LIN {X 0,Y 569.528,Z 1029.936,A -85,B 0,C 180,E1 26173.056,E2 26173.056} C_VEL
LIN {X 0,Y 570.393,Z 1020.294,A -85,B 0,C 180,E1 26170.971,E2 26170.971} C_VEL
LIN {X 0,Y 571.61,Z 1008.72,A -85,B 0,C 180,E1 26168.771,E2 26168.771} C_VEL
LIN {X 0,Y 573.314,Z 993.99,A -85,B 0,C 180,E1 26166.351,E2 26166.351} C_VEL
LIN {X 0,Y 575.02,Z 980.852,A -85,B 0,C 180,E1 26164.454,E2 26164.454} C_VEL
LIN {X 0,Y 577.029,Z 966.146,A -85,B 0,C 180,E1 26162.553,E2 26162.553} C_VEL
LIN {X 0,Y 579.743,Z 946.853,A -85,B 0,C 180,E1 26160.373,E2 26160.373} C_VEL
LIN {X 0,Y 582.096,Z 930.583,A -85,B 0,C 180,E1 26158.751,E2 26158.751} C_VEL
LIN {X 0,Y 584.678,Z 912.881,A -85,B 0,C 180,E1 26157.172,E2 26157.172} C_VEL
LIN {X 0,Y 587.865,Z 890.248,A -85,B 0,C 180,E1 26155.41,E2 26155.41} C_VEL
LIN {X 0,Y 590.454,Z 871.427,A -85,B 0,C 180,E1 26154.132,E2 26154.132} C_VEL
LIN {X 0,Y 593.347,Z 849.656,A -85,B 0,C 180,E1 26152.834,E2 26152.834} C_VEL
LIN {X 0,Y 596.171,Z 826.041,A -85,B 0,C 180,E1 26151.643,E2 26151.643} C_VEL
LIN {X 0,Y 598.242,Z 806.976,A -85,B 0,C 180,E1 26150.819,E2 26150.819} C_VEL
LIN {X 0,Y 600.276,Z 786.144,A -85,B 0,C 180,E1 26150.049,E2 26150.049} C_VEL
LIN {X 0,Y 602.478,Z 760.102,A -85,B 0,C 180,E1 26149.27,E2 26149.27} C_VEL
LIN {X 0,Y 603.931,Z 737.618,A -85,B 0,C 180,E1 26148.757,E2 26148.757} C_VEL
LIN {X 0,Y 604.964,Z 715.893,A -85,B 0,C 180,E1 26148.38,E2 26148.38} C_VEL
LIN {X 0,Y 610.807,Z 481.076,A -85,B 0,C 180,E1 26145.176,E2 26145.176} C_VEL
LIN {X 0,Y 614.185,Z 345.469,A -85,B 0,C 180,E1 26143.295,E2 26143.295} C_VEL
LIN {X 0,Y 598.706,Z 321.323,A -85,B 0,C 180,E1 26141.34,E2 26141.34} C_VEL
LIN {X 0,Y 585.115,Z 301.426,A -85,B 0,C 180,E1 26139.504,E2 26139.504} C_VEL
LIN {X 0,Y 575.623,Z 288.007,A -85,B 0,C 180,E1 26138.136,E2 26138.136} C_VEL
LIN {X 0,Y 573.982,Z 285.549,A -85,B 0,C 180,E1 26137.821,E2 26137.821} C_VEL
LIN {X 0,Y 570.798,Z 278.728,A -85,B 0,C 180,E1 26136.68,E2 26136.68} C_VEL
LIN {X 0,Y 569.328,Z 275.166,A -85,B 0,C 180,E1 26136.04,E2 26136.04} C_VEL
LIN {X 0,Y 569.375,Z 275.014,A -85,B 0,C 180,E1 26132.864,E2 26132.864} C_VEL
LIN {X 0,Y 569.308,Z 275.021,A -85,B 0,C 180,E1 26129.805,E2 26129.805} C_VEL
LIN {X 0,Y 569.365,Z 275.04,A -85,B 0,C 180,E1 26126.604,E2 26126.604} C_VEL
LIN {X 0,Y 569.315,Z 275.047,A -85,B 0,C 180,E1 26123.496,E2 26123.496} C_VEL
LIN {X 0,Y 569.337,Z 275.044,A -85,B 0,C 180,E1 26120.242,E2 26120.242} C_VEL
LIN {X 0,Y 569.33,Z 275.049,A -85,B 0,C 180,E1 26117.161,E2 26117.161} C_VEL
LIN {X 0,Y 569.315,Z 275.058,A -85,B 0,C 180,E1 26113.819,E2 26113.819} C_VEL
LIN {X 0,Y 569.363,Z 275.057,A -85,B 0,C 180,E1 26110.728,E2 26110.728} C_VEL
LIN {X 0,Y 569.31,Z 275.052,A -85,B 0,C 180,E1 26107.569,E2 26107.569} C_VEL
LIN {X 0,Y 569.374,Z 275.038,A -85,B 0,C 180,E1 26104.432,E2 26104.432} C_VEL
LIN {X 0,Y 569.31,Z 275.06,A -85,B 0,C 180,E1 26101.308,E2 26101.308} C_VEL
LIN {X 0,Y 569.37,Z 275.055,A -85,B 0,C 180,E1 26098.189,E2 26098.189} C_VEL
LIN {X 0,Y 569.312,Z 275.045,A -85,B 0,C 180,E1 26095.063,E2 26095.063} C_VEL
LIN {X 0,Y 569.341,Z 275.041,A -85,B 0,C 180,E1 26091.822,E2 26091.822} C_VEL
LIN {X 0,Y 569.326,Z 275.062,A -85,B 0,C 180,E1 26088.758,E2 26088.758} C_VEL
LIN {X 0,Y 569.318,Z 275.065,A -85,B 0,C 180,E1 26085.401,E2 26085.401} C_VEL
LIN {X 0,Y 569.356,Z 275.041,A -85,B 0,C 180,E1 26082.313,E2 26082.313} C_VEL
LIN {X 0,Y 569.31,Z 275.043,A -85,B 0,C 180,E1 26079.112,E2 26079.112} C_VEL
LIN {X 0,Y 569.372,Z 275.038,A -85,B 0,C 180,E1 26076.067,E2 26076.067} C_VEL
LIN {X 0,Y 569.302,Z 274.992,A -85,B 0,C 180,E1 26072.829,E2 26072.829} C_VEL
LIN {X 0,Y 569.376,Z 275.054,A -85,B 0,C 180,E1 26069.734,E2 26069.734} C_VEL
LIN {X 0,Y 569.309,Z 274.991,A -85,B 0,C 180,E1 26066.531,E2 26066.531} C_VEL
LIN {X 0,Y 569.327,Z 275.051,A -85,B 0,C 180,E1 26063.21,E2 26063.21} C_VEL
LIN {X 0,Y 569.336,Z 275.11,A -85,B 0,C 180,E1 26060.201,E2 26060.201} C_VEL
LIN {X 0,Y 570.614,Z 278.424,A -85,B 0,C 180,E1 26059.582,E2 26059.582} C_VEL
LIN {X 0,Y 571.787,Z 280.362,A -85,B 0,C 180,E1 26059.303,E2 26059.303} C_VEL
LIN {X 0,Y 575.084,Z 284.719,A -85,B 0,C 180,E1 26058.812,E2 26058.812} C_VEL
LIN {X 0,Y 589.505,Z 304.979,A -85,B 0,C 180,E1 26056.761,E2 26056.761} C_VEL
LIN {X 0,Y 601.117,Z 322.104,A -85,B 0,C 180,E1 26055.215,E2 26055.215} C_VEL
LIN {X 0,Y 614.233,Z 342.476,A -85,B 0,C 180,E1 26053.57,E2 26053.57} C_VEL
LIN {X 0,Y 609.182,Z 540.418,A -85,B 0,C 180,E1 26050.843,E2 26050.843} C_VEL
LIN {X 0,Y 608.261,Z 548.118,A -85,B 0,C 180,E1 26050.802,E2 26050.802} C_VEL
LIN {X 0,Y 603.163,Z 568.707,A -85,B 0,C 180,E1 26050.927,E2 26050.927} C_VEL
LIN {X 0,Y 602.444,Z 575.314,A -85,B 0,C 180,E1 26050.885,E2 26050.885} C_VEL
LIN {X 0,Y 598.824,Z 711.721,A -85,B 0,C 180,E1 26049.003,E2 26049.003} C_VEL
LIN {X 0,Y 597.3,Z 738.812,A -85,B 0,C 180,E1 26048.485,E2 26048.485} C_VEL
LIN {X 0,Y 595.509,Z 762.096,A -85,B 0,C 180,E1 26047.873,E2 26047.873} C_VEL
LIN {X 0,Y 593.502,Z 784.135,A -85,B 0,C 180,E1 26047.155,E2 26047.155} C_VEL
LIN {X 0,Y 590.692,Z 810.488,A -85,B 0,C 180,E1 26046.091,E2 26046.091} C_VEL
LIN {X 0,Y 588.249,Z 830.386,A -85,B 0,C 180,E1 26045.131,E2 26045.131} C_VEL
LIN {X 0,Y 585.686,Z 849.812,A -85,B 0,C 180,E1 26044.053,E2 26044.053} C_VEL
LIN {X 0,Y 582.368,Z 873.343,A -85,B 0,C 180,E1 26042.539,E2 26042.539} C_VEL
LIN {X 0,Y 579.492,Z 892.375,A -85,B 0,C 180,E1 26041.122,E2 26041.122} C_VEL
LIN {X 0,Y 576.819,Z 909.782,A -85,B 0,C 180,E1 26039.663,E2 26039.663} C_VEL
LIN {X 0,Y 573.672,Z 930.084,A -85,B 0,C 180,E1 26037.734,E2 26037.734} C_VEL
LIN {X 0,Y 571.147,Z 946.426,A -85,B 0,C 180,E1 26035.955,E2 26035.955} C_VEL
LIN {X 0,Y 568.951,Z 961.1,A -85,B 0,C 180,E1 26034.172,E2 26034.172} C_VEL
LIN {X 0,Y 566.637,Z 977.255,A -85,B 0,C 180,E1 26031.968,E2 26031.968} C_VEL
LIN {X 0,Y 564.777,Z 991.296,A -85,B 0,C 180,E1 26029.764,E2 26029.764} C_VEL
LIN {X 0,Y 563.414,Z 1002.582,A -85,B 0,C 180,E1 26027.773,E2 26027.773} C_VEL
LIN {X 0,Y 562.168,Z 1014.61,A -85,B 0,C 180,E1 26025.368,E2 26025.368} C_VEL
LIN {X 0,Y 561.216,Z 1025.111,A -85,B 0,C 180,E1 26022.868,E2 26022.868} C_VEL
LIN {X 0,Y 560.704,Z 1032.614,A -85,B 0,C 180,E1 26020.792,E2 26020.792} C_VEL
LIN {X 0,Y 560.275,Z 1040.198,A -85,B 0,C 180,E1 26018.311,E2 26018.311} C_VEL
LIN {X 0,Y 560.033,Z 1046.307,A -85,B 0,C 180,E1 26015.738,E2 26015.738} C_VEL
LIN {X 0,Y 559.954,Z 1050.223,A -85,B 0,C 180,E1 26013.583,E2 26013.583} C_VEL
LIN {X 0,Y 559.903,Z 1053.047,A -85,B 0,C 180,E1 26011.433,E2 26011.433} C_VEL
LIN {X 0,Y 559.908,Z 1054.995,A -85,B 0,C 180,E1 26008.977,E2 26008.977} C_VEL
LIN {X 0,Y 559.892,Z 1055.388,A -85,B 0,C 180,E1 26006.416,E2 26006.416} C_VEL
LIN {X 0,Y 559.915,Z 1054.551,A -85,B 0,C 180,E1 26004.261,E2 26004.261} C_VEL
LIN {X 0,Y 559.907,Z 1052.74,A -85,B 0,C 180,E1 26002.2,E2 26002.2} C_VEL
LIN {X 0,Y 559.967,Z 1049.596,A -85,B 0,C 180,E1 25999.922,E2 25999.922} C_VEL
LIN {X 0,Y 560.103,Z 1044.215,A -85,B 0,C 180,E1 25997.211,E2 25997.211} C_VEL
LIN {X 0,Y 560.378,Z 1038.165,A -85,B 0,C 180,E1 25994.9,E2 25994.9} C_VEL
LIN {X 0,Y 560.79,Z 1031.129,A -85,B 0,C 180,E1 25992.677,E2 25992.677} C_VEL
LIN {X 0,Y 561.572,Z 1020.991,A -85,B 0,C 180,E1 25990.01,E2 25990.01} C_VEL
LIN {X 0,Y 562.532,Z 1010.781,A -85,B 0,C 180,E1 25987.753,E2 25987.753} C_VEL
LIN {X 0,Y 563.698,Z 1000.216,A -85,B 0,C 180,E1 25985.7,E2 25985.7} C_VEL
LIN {X 0,Y 565.513,Z 985.511,A -85,B 0,C 180,E1 25983.201,E2 25983.201} C_VEL
LIN {X 0,Y 567.441,Z 971.489,A -85,B 0,C 180,E1 25981.131,E2 25981.131} C_VEL
LIN {X 0,Y 569.484,Z 957.456,A -85,B 0,C 180,E1 25979.274,E2 25979.274} C_VEL
LIN {X 0,Y 572.415,Z 938.223,A -85,B 0,C 180,E1 25977.035,E2 25977.035} C_VEL
LIN {X 0,Y 574.992,Z 921.578,A -85,B 0,C 180,E1 25975.339,E2 25975.339} C_VEL
LIN {X 0,Y 577.583,Z 904.918,A -85,B 0,C 180,E1 25973.82,E2 25973.82} C_VEL
LIN {X 0,Y 580.874,Z 883.291,A -85,B 0,C 180,E1 25972.083,E2 25972.083} C_VEL
LIN {X 0,Y 583.821,Z 863.031,A -85,B 0,C 180,E1 25970.678,E2 25970.678} C_VEL
LIN {X 0,Y 586.657,Z 842.71,A -85,B 0,C 180,E1 25969.442,E2 25969.442} C_VEL
LIN {X 0,Y 589.839,Z 817.959,A -85,B 0,C 180,E1 25968.16,E2 25968.16} C_VEL
LIN {X 0,Y 592.189,Z 797.521,A -85,B 0,C 180,E1 25967.264,E2 25967.264} C_VEL
LIN {X 0,Y 594.25,Z 777.464,A -85,B 0,C 180,E1 25966.514,E2 25966.514} C_VEL
LIN {X 0,Y 596.578,Z 751.419,A -85,B 0,C 180,E1 25965.722,E2 25965.722} C_VEL
LIN {X 0,Y 598.111,Z 728.952,A -85,B 0,C 180,E1 25965.2,E2 25965.2} C_VEL
LIN {X 0,Y 599.204,Z 707.344,A -85,B 0,C 180,E1 25964.818,E2 25964.818} C_VEL
LIN {X 0,Y 605.825,Z 470.078,A -85,B 0,C 180,E1 25961.519,E2 25961.519} C_VEL
LIN {X 0,Y 609.288,Z 345.786,A -85,B 0,C 180,E1 25959.748,E2 25959.748} C_VEL
LIN {X 0,Y 596.939,Z 326.269,A -85,B 0,C 180,E1 25958.04,E2 25958.04} C_VEL
LIN {X 0,Y 582.975,Z 306.239,A -85,B 0,C 180,E1 25955.976,E2 25955.976} C_VEL
LIN {X 0,Y 575.262,Z 295.929,A -85,B 0,C 180,E1 25954.758,E2 25954.758} C_VEL
LIN {X 0,Y 570.969,Z 290.29,A -85,B 0,C 180,E1 25954.053,E2 25954.053} C_VEL
LIN {X 0,Y 567.524,Z 285.647,A -85,B 0,C 180,E1 25953.467,E2 25953.467} C_VEL
LIN {X 0,Y 564.242,Z 281.388,A -85,B 0,C 180,E1 25952.898,E2 25952.898} C_VEL
LIN {X 0,Y 562.325,Z 278.884,A -85,B 0,C 180,E1 25952.48,E2 25952.48} C_VEL
LIN {X 0,Y 561.444,Z 276.206,A -85,B 0,C 180,E1 25951.934,E2 25951.934} C_VEL
LIN {X 0,Y 561.373,Z 276.043,A -85,B 0,C 180,E1 25948.978,E2 25948.978} C_VEL
LIN {X 0,Y 561.403,Z 275.99,A -85,B 0,C 180,E1 25945.759,E2 25945.759} C_VEL
LIN {X 0,Y 561.383,Z 276.054,A -85,B 0,C 180,E1 25942.689,E2 25942.689} C_VEL
LIN {X 0,Y 561.372,Z 275.997,A -85,B 0,C 180,E1 25939.239,E2 25939.239} C_VEL
LIN {X 0,Y 561.423,Z 276.037,A -85,B 0,C 180,E1 25936.131,E2 25936.131} C_VEL
LIN {X 0,Y 561.365,Z 275.993,A -85,B 0,C 180,E1 25932.969,E2 25932.969} C_VEL
LIN {X 0,Y 561.435,Z 276.039,A -85,B 0,C 180,E1 25929.741,E2 25929.741} C_VEL
LIN {X 0,Y 561.364,Z 275.982,A -85,B 0,C 180,E1 25926.648,E2 25926.648} C_VEL
LIN {X 0,Y 561.409,Z 276.047,A -85,B 0,C 180,E1 25923.369,E2 25923.369} C_VEL
LIN {X 0,Y 561.374,Z 275.984,A -85,B 0,C 180,E1 25920.306,E2 25920.306} C_VEL
LIN {X 0,Y 561.383,Z 276.051,A -85,B 0,C 180,E1 25916.937,E2 25916.937} C_VEL
LIN {X 0,Y 561.416,Z 275.981,A -85,B 0,C 180,E1 25913.763,E2 25913.763} C_VEL
LIN {X 0,Y 561.37,Z 276.036,A -85,B 0,C 180,E1 25910.569,E2 25910.569} C_VEL
LIN {X 0,Y 561.429,Z 275.989,A -85,B 0,C 180,E1 25907.346,E2 25907.346} C_VEL
LIN {X 0,Y 561.369,Z 276.019,A -85,B 0,C 180,E1 25904.292,E2 25904.292} C_VEL
LIN {X 0,Y 561.41,Z 276.002,A -85,B 0,C 180,E1 25901.036,E2 25901.036} C_VEL
LIN {X 0,Y 561.381,Z 276.02,A -85,B 0,C 180,E1 25897.925,E2 25897.925} C_VEL
LIN {X 0,Y 561.381,Z 276.036,A -85,B 0,C 180,E1 25894.559,E2 25894.559} C_VEL
LIN {X 0,Y 561.414,Z 276.032,A -85,B 0,C 180,E1 25891.49,E2 25891.49} C_VEL
LIN {X 0,Y 561.368,Z 275.993,A -85,B 0,C 180,E1 25888.302,E2 25888.302} C_VEL
LIN {X 0,Y 561.409,Z 276.234,A -85,B 0,C 180,E1 25885.778,E2 25885.778} C_VEL
LIN {X 0,Y 563.065,Z 279.972,A -85,B 0,C 180,E1 25884.999,E2 25884.999} C_VEL
LIN {X 0,Y 566.244,Z 286.174,A -85,B 0,C 180,E1 25883.813,E2 25883.813} C_VEL
LIN {X 0,Y 577.941,Z 302.001,A -85,B 0,C 180,E1 25881.856,E2 25881.856} C_VEL
LIN {X 0,Y 588.085,Z 316.172,A -85,B 0,C 180,E1 25880.292,E2 25880.292} C_VEL
LIN {X 0,Y 599.299,Z 332.935,A -85,B 0,C 180,E1 25878.662,E2 25878.662} C_VEL
LIN {X 0,Y 609.505,Z 349.548,A -85,B 0,C 180,E1 25877.259,E2 25877.259} C_VEL
LIN {X 0,Y 602.826,Z 581.277,A -85,B 0,C 180,E1 25874.013,E2 25874.013} C_VEL
LIN {X 0,Y 598.937,Z 720.481,A -85,B 0,C 180,E1 25872.074,E2 25872.074} C_VEL
LIN {X 0,Y 597.342,Z 747.614,A -85,B 0,C 180,E1 25871.554,E2 25871.554} C_VEL
LIN {X 0,Y 595.485,Z 771.005,A -85,B 0,C 180,E1 25870.937,E2 25870.937} C_VEL
LIN {X 0,Y 593.458,Z 792.738,A -85,B 0,C 180,E1 25870.227,E2 25870.227} C_VEL
LIN {X 0,Y 590.584,Z 819.273,A -85,B 0,C 180,E1 25869.157,E2 25869.157} C_VEL
LIN {X 0,Y 588.069,Z 839.646,A -85,B 0,C 180,E1 25868.174,E2 25868.174} C_VEL
LIN {X 0,Y 585.356,Z 860.369,A -85,B 0,C 180,E1 25867.022,E2 25867.022} C_VEL
LIN {X 0,Y 581.977,Z 884.248,A -85,B 0,C 180,E1 25865.474,E2 25865.474} C_VEL
LIN {X 0,Y 579.28,Z 902.355,A -85,B 0,C 180,E1 25864.123,E2 25864.123} C_VEL
LIN {X 0,Y 576.588,Z 920.113,A -85,B 0,C 180,E1 25862.637,E2 25862.637} C_VEL
LIN {X 0,Y 573.347,Z 941.298,A -85,B 0,C 180,E1 25860.613,E2 25860.613} C_VEL
LIN {X 0,Y 570.932,Z 957.248,A -85,B 0,C 180,E1 25858.876,E2 25858.876} C_VEL
LIN {X 0,Y 568.653,Z 972.852,A -85,B 0,C 180,E1 25856.978,E2 25856.978} C_VEL
LIN {X 0,Y 566.284,Z 989.784,A -85,B 0,C 180,E1 25854.627,E2 25854.627} C_VEL
LIN {X 0,Y 564.612,Z 1002.542,A -85,B 0,C 180,E1 25852.6,E2 25852.6} C_VEL
LIN {X 0,Y 563.112,Z 1015.592,A -85,B 0,C 180,E1 25850.258,E2 25850.258} C_VEL
LIN {X 0,Y 561.91,Z 1027.179,A -85,B 0,C 180,E1 25847.822,E2 25847.822} C_VEL
LIN {X 0,Y 561.157,Z 1035.877,A -85,B 0,C 180,E1 25845.714,E2 25845.714} C_VEL
LIN {X 0,Y 560.633,Z 1043.715,A -85,B 0,C 180,E1 25843.511,E2 25843.511} C_VEL
LIN {X 0,Y 560.216,Z 1051.623,A -85,B 0,C 180,E1 25840.801,E2 25840.801} C_VEL
LIN {X 0,Y 560.022,Z 1056.828,A -85,B 0,C 180,E1 25838.522,E2 25838.522} C_VEL
LIN {X 0,Y 559.955,Z 1060.486,A -85,B 0,C 180,E1 25836.459,E2 25836.459} C_VEL
LIN {X 0,Y 559.914,Z 1063.47,A -85,B 0,C 180,E1 25834.096,E2 25834.096} C_VEL
LIN {X 0,Y 559.9,Z 1065.19,A -85,B 0,C 180,E1 25831.433,E2 25831.433} C_VEL
LIN {X 0,Y 559.898,Z 1065.349,A -85,B 0,C 180,E1 25829.284,E2 25829.284} C_VEL
LIN {X 0,Y 559.913,Z 1064.436,A -85,B 0,C 180,E1 25827.134,E2 25827.134} C_VEL
LIN {X 0,Y 559.918,Z 1062.446,A -85,B 0,C 180,E1 25824.98,E2 25824.98} C_VEL
LIN {X 0,Y 559.999,Z 1058.461,A -85,B 0,C 180,E1 25822.294,E2 25822.294} C_VEL
LIN {X 0,Y 560.127,Z 1053.403,A -85,B 0,C 180,E1 25819.925,E2 25819.925} C_VEL
LIN {X 0,Y 560.387,Z 1047.876,A -85,B 0,C 180,E1 25817.846,E2 25817.846} C_VEL
LIN {X 0,Y 560.832,Z 1040.535,A -85,B 0,C 180,E1 25815.546,E2 25815.546} C_VEL
LIN {X 0,Y 561.656,Z 1029.935,A -85,B 0,C 180,E1 25812.811,E2 25812.811} C_VEL
LIN {X 0,Y 562.582,Z 1020.281,A -85,B 0,C 180,E1 25810.694,E2 25810.694} C_VEL
LIN {X 0,Y 563.89,Z 1008.718,A -85,B 0,C 180,E1 25808.466,E2 25808.466} C_VEL
LIN {X 0,Y 565.711,Z 993.988,A -85,B 0,C 180,E1 25806.014,E2 25806.014} C_VEL
LIN {X 0,Y 567.513,Z 980.818,A -85,B 0,C 180,E1 25804.091,E2 25804.091} C_VEL
LIN {X 0,Y 569.76,Z 965.215,A -85,B 0,C 180,E1 25802.059,E2 25802.059} C_VEL
LIN {X 0,Y 572.576,Z 946.397,A -85,B 0,C 180,E1 25799.922,E2 25799.922} C_VEL
LIN {X 0,Y 575.002,Z 930.5,A -85,B 0,C 180,E1 25798.321,E2 25798.321} C_VEL
LIN {X 0,Y 577.81,Z 912.188,A -85,B 0,C 180,E1 25796.673,E2 25796.673} C_VEL
LIN {X 0,Y 581.131,Z 889.829,A -85,B 0,C 180,E1 25794.923,E2 25794.923} C_VEL
LIN {X 0,Y 583.806,Z 871.342,A -85,B 0,C 180,E1 25793.659,E2 25793.659} C_VEL
LIN {X 0,Y 586.842,Z 849.57,A -85,B 0,C 180,E1 25792.351,E2 25792.351} C_VEL
LIN {X 0,Y 589.796,Z 825.94,A -85,B 0,C 180,E1 25791.152,E2 25791.152} C_VEL
LIN {X 0,Y 591.962,Z 806.826,A -85,B 0,C 180,E1 25790.321,E2 25790.321} C_VEL
LIN {X 0,Y 594.004,Z 786.663,A -85,B 0,C 180,E1 25789.572,E2 25789.572} C_VEL
LIN {X 0,Y 596.265,Z 761.264,A -85,B 0,C 180,E1 25788.801,E2 25788.801} C_VEL
LIN {X 0,Y 597.85,Z 737.716,A -85,B 0,C 180,E1 25788.258,E2 25788.258} C_VEL
LIN {X 0,Y 598.921,Z 716.111,A -85,B 0,C 180,E1 25787.88,E2 25787.88} C_VEL
LIN {X 0,Y 604.999,Z 482.812,A -85,B 0,C 180,E1 25784.673,E2 25784.673} C_VEL
LIN {X 0,Y 608.49,Z 349.049,A -85,B 0,C 180,E1 25782.803,E2 25782.803} C_VEL
LIN {X 0,Y 593.069,Z 324.968,A -85,B 0,C 180,E1 25780.808,E2 25780.808} C_VEL
LIN {X 0,Y 578.742,Z 303.894,A -85,B 0,C 180,E1 25778.812,E2 25778.812} C_VEL
LIN {X 0,Y 567.989,Z 289.037,A -85,B 0,C 180,E1 25777.207,E2 25777.207} C_VEL
LIN {X 0,Y 565.798,Z 285.613,A -85,B 0,C 180,E1 25776.805,E2 25776.805} C_VEL
LIN {X 0,Y 562.526,Z 279.268,A -85,B 0,C 180,E1 25775.663,E2 25775.663} C_VEL
LIN {X 0,Y 561.444,Z 276.151,A -85,B 0,C 180,E1 25775.098,E2 25775.098} C_VEL
LIN {X 0,Y 561.372,Z 276.039,A -85,B 0,C 180,E1 25771.938,E2 25771.938} C_VEL
LIN {X 0,Y 561.437,Z 275.984,A -85,B 0,C 180,E1 25768.741,E2 25768.741} C_VEL
LIN {X 0,Y 561.379,Z 276.053,A -85,B 0,C 180,E1 25765.533,E2 25765.533} C_VEL
LIN {X 0,Y 561.39,Z 276.053,A -85,B 0,C 180,E1 25762.156,E2 25762.156} C_VEL
LIN {X 0,Y 561.396,Z 276.044,A -85,B 0,C 180,E1 25759.13,E2 25759.13} C_VEL
LIN {X 0,Y 561.374,Z 276.039,A -85,B 0,C 180,E1 25755.814,E2 25755.814} C_VEL
LIN {X 0,Y 561.424,Z 276.028,A -85,B 0,C 180,E1 25752.759,E2 25752.759} C_VEL
LIN {X 0,Y 561.371,Z 276.046,A -85,B 0,C 180,E1 25749.535,E2 25749.535} C_VEL
LIN {X 0,Y 561.438,Z 276.048,A -85,B 0,C 180,E1 25746.339,E2 25746.339} C_VEL
LIN {X 0,Y 561.376,Z 276.042,A -85,B 0,C 180,E1 25743.165,E2 25743.165} C_VEL
LIN {X 0,Y 561.387,Z 276.03,A -85,B 0,C 180,E1 25739.796,E2 25739.796} C_VEL
LIN {X 0,Y 561.399,Z 276.043,A -85,B 0,C 180,E1 25736.733,E2 25736.733} C_VEL
LIN {X 0,Y 561.375,Z 276.052,A -85,B 0,C 180,E1 25733.454,E2 25733.454} C_VEL
LIN {X 0,Y 561.426,Z 276.03,A -85,B 0,C 180,E1 25730.363,E2 25730.363} C_VEL
LIN {X 0,Y 561.368,Z 276.03,A -85,B 0,C 180,E1 25727.135,E2 25727.135} C_VEL
LIN {X 0,Y 561.434,Z 276.032,A -85,B 0,C 180,E1 25723.975,E2 25723.975} C_VEL
LIN {X 0,Y 561.379,Z 276.052,A -85,B 0,C 180,E1 25720.761,E2 25720.761} C_VEL
LIN {X 0,Y 561.382,Z 276.053,A -85,B 0,C 180,E1 25717.311,E2 25717.311} C_VEL
LIN {X 0,Y 561.401,Z 275.973,A -85,B 0,C 180,E1 25714.241,E2 25714.241} C_VEL
LIN {X 0,Y 561.37,Z 276.035,A -85,B 0,C 180,E1 25710.991,E2 25710.991} C_VEL
LIN {X 0,Y 561.425,Z 275.982,A -85,B 0,C 180,E1 25707.945,E2 25707.945} C_VEL
LIN {X 0,Y 561.369,Z 276.023,A -85,B 0,C 180,E1 25704.753,E2 25704.753} C_VEL
LIN {X 0,Y 561.429,Z 276.025,A -85,B 0,C 180,E1 25701.57,E2 25701.57} C_VEL
LIN {X 0,Y 561.421,Z 276.33,A -85,B 0,C 180,E1 25701.064,E2 25701.064} C_VEL
LIN {X 0,Y 562.725,Z 279.607,A -85,B 0,C 180,E1 25700.497,E2 25700.497} C_VEL
LIN {X 0,Y 568.48,Z 287.302,A -85,B 0,C 180,E1 25699.581,E2 25699.581} C_VEL
LIN {X 0,Y 579.175,Z 301.934,A -85,B 0,C 180,E1 25697.995,E2 25697.995} C_VEL
LIN {X 0,Y 592.975,Z 321.874,A -85,B 0,C 180,E1 25696.078,E2 25696.078} C_VEL
LIN {X 0,Y 608.546,Z 345.901,A -85,B 0,C 180,E1 25694.064,E2 25694.064} C_VEL
LIN {X 0,Y 602.665,Z 566.89,A -85,B 0,C 180,E1 25691,E2 25691} C_VEL
LIN {X 0,Y 602.444,Z 575.314,A -85,B 0,C 180,E1 25690.885,E2 25690.885} C_VEL
LIN {X 0,Y 601.525,Z 583.011,A -85,B 0,C 180,E1 25690.844,E2 25690.844} C_VEL
LIN {X 0,Y 596.424,Z 603.594,A -85,B 0,C 180,E1 25690.97,E2 25690.97} C_VEL
LIN {X 0,Y 595.678,Z 610.202,A -85,B 0,C 180,E1 25690.931,E2 25690.931} C_VEL
LIN {X 0,Y 592.806,Z 712.303,A -85,B 0,C 180,E1 25689.507,E2 25689.507} C_VEL
LIN {X 0,Y 591.143,Z 740.202,A -85,B 0,C 180,E1 25688.962,E2 25688.962} C_VEL
LIN {X 0,Y 589.328,Z 762.839,A -85,B 0,C 180,E1 25688.36,E2 25688.36} C_VEL
LIN {X 0,Y 587.139,Z 785.951,A -85,B 0,C 180,E1 25687.596,E2 25687.596} C_VEL
LIN {X 0,Y 584.41,Z 810.278,A -85,B 0,C 180,E1 25686.602,E2 25686.602} C_VEL
LIN {X 0,Y 581.833,Z 830.487,A -85,B 0,C 180,E1 25685.623,E2 25685.623} C_VEL
LIN {X 0,Y 579.156,Z 849.987,A -85,B 0,C 180,E1 25684.535,E2 25684.535} C_VEL
LIN {X 0,Y 575.693,Z 873.47,A -85,B 0,C 180,E1 25683.012,E2 25683.012} C_VEL
LIN {X 0,Y 572.691,Z 892.433,A -85,B 0,C 180,E1 25681.586,E2 25681.586} C_VEL
LIN {X 0,Y 569.895,Z 909.784,A -85,B 0,C 180,E1 25680.118,E2 25680.118} C_VEL
LIN {X 0,Y 566.565,Z 930.101,A -85,B 0,C 180,E1 25678.17,E2 25678.17} C_VEL
LIN {X 0,Y 563.824,Z 946.901,A -85,B 0,C 180,E1 25676.318,E2 25676.318} C_VEL
LIN {X 0,Y 561.5,Z 961.649,A -85,B 0,C 180,E1 25674.499,E2 25674.499} C_VEL
LIN {X 0,Y 558.959,Z 978.32,A -85,B 0,C 180,E1 25672.175,E2 25672.175} C_VEL
LIN {X 0,Y 557.094,Z 991.586,A -85,B 0,C 180,E1 25670.048,E2 25670.048} C_VEL
LIN {X 0,Y 555.579,Z 1003.394,A -85,B 0,C 180,E1 25667.924,E2 25667.924} C_VEL
LIN {X 0,Y 554.167,Z 1016.175,A -85,B 0,C 180,E1 25665.274,E2 25665.274} C_VEL
LIN {X 0,Y 553.309,Z 1025.285,A -85,B 0,C 180,E1 25663.055,E2 25663.055} C_VEL
LIN {X 0,Y 552.734,Z 1033.114,A -85,B 0,C 180,E1 25660.844,E2 25660.844} C_VEL
LIN {X 0,Y 552.272,Z 1040.877,A -85,B 0,C 180,E1 25658.223,E2 25658.223} C_VEL
LIN {X 0,Y 552.036,Z 1046.6,A -85,B 0,C 180,E1 25655.717,E2 25655.717} C_VEL
LIN {X 0,Y 551.957,Z 1050.291,A -85,B 0,C 180,E1 25653.635,E2 25653.635} C_VEL
LIN {X 0,Y 551.903,Z 1053.095,A -85,B 0,C 180,E1 25651.453,E2 25651.453} C_VEL
LIN {X 0,Y 551.908,Z 1055.024,A -85,B 0,C 180,E1 25648.962,E2 25648.962} C_VEL
LIN {X 0,Y 551.893,Z 1055.378,A -85,B 0,C 180,E1 25646.364,E2 25646.364} C_VEL
LIN {X 0,Y 551.915,Z 1054.521,A -85,B 0,C 180,E1 25644.177,E2 25644.177} C_VEL
LIN {X 0,Y 551.912,Z 1052.691,A -85,B 0,C 180,E1 25642.086,E2 25642.086} C_VEL
LIN {X 0,Y 551.977,Z 1049.527,A -85,B 0,C 180,E1 25639.774,E2 25639.774} C_VEL
LIN {X 0,Y 552.123,Z 1044.017,A -85,B 0,C 180,E1 25636.987,E2 25636.987} C_VEL
LIN {X 0,Y 552.409,Z 1038.227,A -85,B 0,C 180,E1 25634.745,E2 25634.745} C_VEL
LIN {X 0,Y 552.844,Z 1031.33,A -85,B 0,C 180,E1 25632.529,E2 25632.529} C_VEL
LIN {X 0,Y 553.649,Z 1021.605,A -85,B 0,C 180,E1 25629.905,E2 25629.905} C_VEL
LIN {X 0,Y 554.698,Z 1011.073,A -85,B 0,C 180,E1 25627.533,E2 25627.533} C_VEL
LIN {X 0,Y 555.938,Z 1000.54,A -85,B 0,C 180,E1 25625.451,E2 25625.451} C_VEL
LIN {X 0,Y 557.87,Z 985.954,A -85,B 0,C 180,E1 25622.919,E2 25622.919} C_VEL
LIN {X 0,Y 559.902,Z 972.006,A -85,B 0,C 180,E1 25620.822,E2 25620.822} C_VEL
LIN {X 0,Y 562.054,Z 958.016,A -85,B 0,C 180,E1 25618.942,E2 25618.942} C_VEL
LIN {X 0,Y 564.988,Z 939.912,A -85,B 0,C 180,E1 25616.788,E2 25616.788} C_VEL
LIN {X 0,Y 567.85,Z 922.304,A -85,B 0,C 180,E1 25614.964,E2 25614.964} C_VEL
LIN {X 0,Y 570.56,Z 905.692,A -85,B 0,C 180,E1 25613.428,E2 25613.428} C_VEL
LIN {X 0,Y 574.012,Z 884.213,A -85,B 0,C 180,E1 25611.675,E2 25611.675} C_VEL
LIN {X 0,Y 577.093,Z 864.052,A -85,B 0,C 180,E1 25610.258,E2 25610.258} C_VEL
LIN {X 0,Y 579.998,Z 844.262,A -85,B 0,C 180,E1 25609.034,E2 25609.034} C_VEL
LIN {X 0,Y 583.387,Z 819.502,A -85,B 0,C 180,E1 25607.723,E2 25607.723} C_VEL
LIN {X 0,Y 585.857,Z 799.097,A -85,B 0,C 180,E1 25606.812,E2 25606.812} C_VEL
LIN {X 0,Y 588.053,Z 778.788,A -85,B 0,C 180,E1 25606.04,E2 25606.04} C_VEL
LIN {X 0,Y 590.445,Z 753.849,A -85,B 0,C 180,E1 25605.26,E2 25605.26} C_VEL
LIN {X 0,Y 592.19,Z 729.486,A -85,B 0,C 180,E1 25604.684,E2 25604.684} C_VEL
LIN {X 0,Y 593.34,Z 707.825,A -85,B 0,C 180,E1 25604.297,E2 25604.297} C_VEL
LIN {X 0,Y 600.267,Z 471.875,A -85,B 0,C 180,E1 25600.989,E2 25600.989} C_VEL
LIN {X 0,Y 603.887,Z 349.551,A -85,B 0,C 180,E1 25599.235,E2 25599.235} C_VEL
LIN {X 0,Y 591.822,Z 330.448,A -85,B 0,C 180,E1 25597.522,E2 25597.522} C_VEL
LIN {X 0,Y 578.691,Z 311.617,A -85,B 0,C 180,E1 25595.532,E2 25595.532} C_VEL
LIN {X 0,Y 571.67,Z 302.16,A -85,B 0,C 180,E1 25594.399,E2 25594.399} C_VEL
LIN {X 0,Y 564.132,Z 292.127,A -85,B 0,C 180,E1 25593.117,E2 25593.117} C_VEL
LIN {X 0,Y 556.065,Z 282.011,A -85,B 0,C 180,E1 25591.673,E2 25591.673} C_VEL
LIN {X 0,Y 553.925,Z 278.958,A -85,B 0,C 180,E1 25591.173,E2 25591.173} C_VEL
LIN {X 0,Y 553.457,Z 277.112,A -85,B 0,C 180,E1 25590.749,E2 25590.749} C_VEL
LIN {X 0,Y 553.439,Z 277.008,A -85,B 0,C 180,E1 25587.433,E2 25587.433} C_VEL
LIN {X 0,Y 553.485,Z 276.999,A -85,B 0,C 180,E1 25584.21,E2 25584.21} C_VEL
LIN {X 0,Y 553.429,Z 276.99,A -85,B 0,C 180,E1 25581.072,E2 25581.072} C_VEL
LIN {X 0,Y 553.492,Z 277.017,A -85,B 0,C 180,E1 25577.819,E2 25577.819} C_VEL
LIN {X 0,Y 553.431,Z 276.983,A -85,B 0,C 180,E1 25574.652,E2 25574.652} C_VEL
LIN {X 0,Y 553.447,Z 277.026,A -85,B 0,C 180,E1 25571.252,E2 25571.252} C_VEL
LIN {X 0,Y 553.466,Z 276.976,A -85,B 0,C 180,E1 25568.106,E2 25568.106} C_VEL
LIN {X 0,Y 553.432,Z 277.011,A -85,B 0,C 180,E1 25564.871,E2 25564.871} C_VEL
LIN {X 0,Y 553.495,Z 276.989,A -85,B 0,C 180,E1 25561.656,E2 25561.656} C_VEL
LIN {X 0,Y 553.429,Z 276.992,A -85,B 0,C 180,E1 25558.551,E2 25558.551} C_VEL
LIN {X 0,Y 553.479,Z 277.02,A -85,B 0,C 180,E1 25555.337,E2 25555.337} C_VEL
LIN {X 0,Y 553.433,Z 276.972,A -85,B 0,C 180,E1 25552.212,E2 25552.212} C_VEL
LIN {X 0,Y 553.444,Z 277.031,A -85,B 0,C 180,E1 25548.818,E2 25548.818} C_VEL
LIN {X 0,Y 553.473,Z 276.965,A -85,B 0,C 180,E1 25545.67,E2 25545.67} C_VEL
LIN {X 0,Y 553.436,Z 277.038,A -85,B 0,C 180,E1 25542.439,E2 25542.439} C_VEL
LIN {X 0,Y 553.486,Z 276.97,A -85,B 0,C 180,E1 25539.152,E2 25539.152} C_VEL
LIN {X 0,Y 553.441,Z 277.035,A -85,B 0,C 180,E1 25536.015,E2 25536.015} C_VEL
LIN {X 0,Y 553.448,Z 277.031,A -85,B 0,C 180,E1 25532.568,E2 25532.568} C_VEL
LIN {X 0,Y 553.469,Z 277.018,A -85,B 0,C 180,E1 25529.512,E2 25529.512} C_VEL
LIN {X 0,Y 553.516,Z 277.224,A -85,B 0,C 180,E1 25526.907,E2 25526.907} C_VEL
LIN {X 0,Y 554.911,Z 280.716,A -85,B 0,C 180,E1 25526.166,E2 25526.166} C_VEL
LIN {X 0,Y 555.996,Z 282.63,A -85,B 0,C 180,E1 25525.744,E2 25525.744} C_VEL
LIN {X 0,Y 557.985,Z 286.163,A -85,B 0,C 180,E1 25525.041,E2 25525.041} C_VEL
LIN {X 0,Y 561.744,Z 291.309,A -85,B 0,C 180,E1 25524.342,E2 25524.342} C_VEL
LIN {X 0,Y 573.758,Z 307.294,A -85,B 0,C 180,E1 25522.304,E2 25522.304} C_VEL
LIN {X 0,Y 586.234,Z 325.024,A -85,B 0,C 180,E1 25520.348,E2 25520.348} C_VEL
LIN {X 0,Y 599.098,Z 344.785,A -85,B 0,C 180,E1 25518.47,E2 25518.47} C_VEL
LIN {X 0,Y 604.058,Z 353.409,A -85,B 0,C 180,E1 25517.771,E2 25517.771} C_VEL
LIN {X 0,Y 597.06,Z 584.784,A -85,B 0,C 180,E1 25514.507,E2 25514.507} C_VEL
LIN {X 0,Y 593.074,Z 720.392,A -85,B 0,C 180,E1 25512.602,E2 25512.602} C_VEL
LIN {X 0,Y 591.425,Z 747.357,A -85,B 0,C 180,E1 25512.083,E2 25512.083} C_VEL
LIN {X 0,Y 589.478,Z 770.851,A -85,B 0,C 180,E1 25511.461,E2 25511.461} C_VEL
LIN {X 0,Y 587.313,Z 793.026,A -85,B 0,C 180,E1 25510.732,E2 25510.732} C_VEL
LIN {X 0,Y 584.316,Z 819.274,A -85,B 0,C 180,E1 25509.664,E2 25509.664} C_VEL
LIN {X 0,Y 581.684,Z 839.571,A -85,B 0,C 180,E1 25508.677,E2 25508.677} C_VEL
LIN {X 0,Y 578.7,Z 861.221,A -85,B 0,C 180,E1 25507.459,E2 25507.459} C_VEL
LIN {X 0,Y 575.269,Z 884.205,A -85,B 0,C 180,E1 25505.947,E2 25505.947} C_VEL
LIN {X 0,Y 572.446,Z 902.267,A -85,B 0,C 180,E1 25504.588,E2 25504.588} C_VEL
LIN {X 0,Y 569.62,Z 920.025,A -85,B 0,C 180,E1 25503.087,E2 25503.087} C_VEL
LIN {X 0,Y 566.182,Z 941.211,A -85,B 0,C 180,E1 25501.043,E2 25501.043} C_VEL
LIN {X 0,Y 563.605,Z 957.386,A -85,B 0,C 180,E1 25499.259,E2 25499.259} C_VEL
LIN {X 0,Y 561.113,Z 973.615,A -85,B 0,C 180,E1 25497.256,E2 25497.256} C_VEL
LIN {X 0,Y 558.709,Z 989.708,A -85,B 0,C 180,E1 25494.983,E2 25494.983} C_VEL
LIN {X 0,Y 556.957,Z 1002.531,A -85,B 0,C 180,E1 25492.928,E2 25492.928} C_VEL
LIN {X 0,Y 555.402,Z 1015.017,A -85,B 0,C 180,E1 25490.662,E2 25490.662} C_VEL
LIN {X 0,Y 554.063,Z 1027.177,A -85,B 0,C 180,E1 25488.083,E2 25488.083} C_VEL
LIN {X 0,Y 553.257,Z 1035.876,A -85,B 0,C 180,E1 25485.944,E2 25485.944} C_VEL
LIN {X 0,Y 552.694,Z 1043.714,A -85,B 0,C 180,E1 25483.709,E2 25483.709} C_VEL
LIN {X 0,Y 552.237,Z 1051.623,A -85,B 0,C 180,E1 25480.959,E2 25480.959} C_VEL
LIN {X 0,Y 552.03,Z 1056.828,A -85,B 0,C 180,E1 25478.646,E2 25478.646} C_VEL
LIN {X 0,Y 551.959,Z 1060.486,A -85,B 0,C 180,E1 25476.553,E2 25476.553} C_VEL
LIN {X 0,Y 551.912,Z 1063.47,A -85,B 0,C 180,E1 25474.156,E2 25474.156} C_VEL
LIN {X 0,Y 551.899,Z 1065.19,A -85,B 0,C 180,E1 25471.453,E2 25471.453} C_VEL
LIN {X 0,Y 551.898,Z 1065.349,A -85,B 0,C 180,E1 25469.273,E2 25469.273} C_VEL
LIN {X 0,Y 551.913,Z 1064.436,A -85,B 0,C 180,E1 25467.092,E2 25467.092} C_VEL
LIN {X 0,Y 551.92,Z 1062.446,A -85,B 0,C 180,E1 25464.907,E2 25464.907} C_VEL
LIN {X 0,Y 552.007,Z 1058.48,A -85,B 0,C 180,E1 25462.192,E2 25462.192} C_VEL
LIN {X 0,Y 552.15,Z 1053.403,A -85,B 0,C 180,E1 25459.778,E2 25459.778} C_VEL
LIN {X 0,Y 552.423,Z 1047.876,A -85,B 0,C 180,E1 25457.668,E2 25457.668} C_VEL
LIN {X 0,Y 552.902,Z 1040.609,A -85,B 0,C 180,E1 25455.357,E2 25455.357} C_VEL
LIN {X 0,Y 553.751,Z 1030.392,A -85,B 0,C 180,E1 25452.667,E2 25452.667} C_VEL
LIN {X 0,Y 554.781,Z 1020.291,A -85,B 0,C 180,E1 25450.414,E2 25450.414} C_VEL
LIN {X 0,Y 556.103,Z 1009.29,A -85,B 0,C 180,E1 25448.26,E2 25448.26} C_VEL
LIN {X 0,Y 558.122,Z 993.935,A -85,B 0,C 180,E1 25445.667,E2 25445.667} C_VEL
LIN {X 0,Y 560.067,Z 980.371,A -85,B 0,C 180,E1 25443.667,E2 25443.667} C_VEL
LIN {X 0,Y 562.55,Z 964.284,A -85,B 0,C 180,E1 25441.553,E2 25441.553} C_VEL
LIN {X 0,Y 565.458,Z 945.829,A -85,B 0,C 180,E1 25439.447,E2 25439.447} C_VEL
LIN {X 0,Y 567.958,Z 930.266,A -85,B 0,C 180,E1 25437.866,E2 25437.866} C_VEL
LIN {X 0,Y 570.993,Z 911.493,A -85,B 0,C 180,E1 25436.161,E2 25436.161} C_VEL
LIN {X 0,Y 574.398,Z 889.744,A -85,B 0,C 180,E1 25434.45,E2 25434.45} C_VEL
LIN {X 0,Y 577.25,Z 870.95,A -85,B 0,C 180,E1 25433.155,E2 25433.155} C_VEL
LIN {X 0,Y 580.374,Z 849.448,A -85,B 0,C 180,E1 25431.857,E2 25431.857} C_VEL
LIN {X 0,Y 583.451,Z 825.738,A -85,B 0,C 180,E1 25430.648,E2 25430.648} C_VEL
LIN {X 0,Y 585.713,Z 806.562,A -85,B 0,C 180,E1 25429.812,E2 25429.812} C_VEL
LIN {X 0,Y 587.765,Z 787.083,A -85,B 0,C 180,E1 25429.084,E2 25429.084} C_VEL
LIN {X 0,Y 590.114,Z 761.902,A -85,B 0,C 180,E1 25428.31,E2 25428.31} C_VEL
LIN {X 0,Y 591.817,Z 737.565,A -85,B 0,C 180,E1 25427.745,E2 25427.745} C_VEL
LIN {X 0,Y 592.923,Z 715.981,A -85,B 0,C 180,E1 25427.366,E2 25427.366} C_VEL
LIN {X 0,Y 599.278,Z 482.934,A -85,B 0,C 180,E1 25424.139,E2 25424.139} C_VEL
LIN {X 0,Y 602.823,Z 352.644,A -85,B 0,C 180,E1 25422.3,E2 25422.3} C_VEL
LIN {X 0,Y 587.198,Z 328.136,A -85,B 0,C 180,E1 25420.225,E2 25420.225} C_VEL
LIN {X 0,Y 574.36,Z 309.352,A -85,B 0,C 180,E1 25418.394,E2 25418.394} C_VEL
LIN {X 0,Y 564.696,Z 295.759,A -85,B 0,C 180,E1 25416.92,E2 25416.92} C_VEL
LIN {X 0,Y 560.206,Z 289.836,A -85,B 0,C 180,E1 25416.213,E2 25416.213} C_VEL
LIN {X 0,Y 557.668,Z 285.939,A -85,B 0,C 180,E1 25415.769,E2 25415.769} C_VEL
LIN {X 0,Y 555.649,Z 281.85,A -85,B 0,C 180,E1 25415.033,E2 25415.033} C_VEL
LIN {X 0,Y 553.664,Z 278.107,A -85,B 0,C 180,E1 25414.295,E2 25414.295} C_VEL
LIN {X 0,Y 553.448,Z 277.12,A -85,B 0,C 180,E1 25414.06,E2 25414.06} C_VEL
LIN {X 0,Y 553.506,Z 277.022,A -85,B 0,C 180,E1 25410.866,E2 25410.866} C_VEL
LIN {X 0,Y 553.433,Z 276.987,A -85,B 0,C 180,E1 25407.667,E2 25407.667} C_VEL
LIN {X 0,Y 553.461,Z 277.021,A -85,B 0,C 180,E1 25404.325,E2 25404.325} C_VEL
LIN {X 0,Y 553.448,Z 277.032,A -85,B 0,C 180,E1 25401.293,E2 25401.293} C_VEL
LIN {X 0,Y 553.44,Z 277.038,A -85,B 0,C 180,E1 25397.887,E2 25397.887} C_VEL
LIN {X 0,Y 553.507,Z 277.034,A -85,B 0,C 180,E1 25394.65,E2 25394.65} C_VEL
LIN {X 0,Y 553.433,Z 277.033,A -85,B 0,C 180,E1 25391.463,E2 25391.463} C_VEL
LIN {X 0,Y 553.475,Z 277.016,A -85,B 0,C 180,E1 25388.205,E2 25388.205} C_VEL
LIN {X 0,Y 553.438,Z 277.031,A -85,B 0,C 180,E1 25385.183,E2 25385.183} C_VEL
LIN {X 0,Y 553.445,Z 277.039,A -85,B 0,C 180,E1 25381.76,E2 25381.76} C_VEL
LIN {X 0,Y 553.459,Z 277.028,A -85,B 0,C 180,E1 25378.758,E2 25378.758} C_VEL
LIN {X 0,Y 553.432,Z 277.019,A -85,B 0,C 180,E1 25375.44,E2 25375.44} C_VEL
LIN {X 0,Y 553.506,Z 277.018,A -85,B 0,C 180,E1 25372.213,E2 25372.213} C_VEL
LIN {X 0,Y 553.438,Z 277.04,A -85,B 0,C 180,E1 25368.959,E2 25368.959} C_VEL
LIN {X 0,Y 553.45,Z 277.039,A -85,B 0,C 180,E1 25365.548,E2 25365.548} C_VEL
LIN {X 0,Y 553.463,Z 277.017,A -85,B 0,C 180,E1 25362.44,E2 25362.44} C_VEL
LIN {X 0,Y 553.433,Z 277.02,A -85,B 0,C 180,E1 25359.15,E2 25359.15} C_VEL
LIN {X 0,Y 553.497,Z 277.011,A -85,B 0,C 180,E1 25356.017,E2 25356.017} C_VEL
LIN {X 0,Y 553.427,Z 276.964,A -85,B 0,C 180,E1 25352.736,E2 25352.736} C_VEL
LIN {X 0,Y 553.467,Z 277.03,A -85,B 0,C 180,E1 25349.492,E2 25349.492} C_VEL
LIN {X 0,Y 553.444,Z 276.963,A -85,B 0,C 180,E1 25346.313,E2 25346.313} C_VEL
LIN {X 0,Y 553.435,Z 277.024,A -85,B 0,C 180,E1 25342.992,E2 25342.992} C_VEL
LIN {X 0,Y 553.517,Z 277.35,A -85,B 0,C 180,E1 25342.048,E2 25342.048} C_VEL
LIN {X 0,Y 554.749,Z 280.433,A -85,B 0,C 180,E1 25341.55,E2 25341.55} C_VEL
LIN {X 0,Y 561.716,Z 289.465,A -85,B 0,C 180,E1 25340.412,E2 25340.412} C_VEL
LIN {X 0,Y 565.266,Z 294.257,A -85,B 0,C 180,E1 25339.852,E2 25339.852} C_VEL
LIN {X 0,Y 575.183,Z 307.839,A -85,B 0,C 180,E1 25338.356,E2 25338.356} C_VEL
LIN {X 0,Y 589.681,Z 328.978,A -85,B 0,C 180,E1 25336.309,E2 25336.309} C_VEL
LIN {X 0,Y 602.899,Z 349.758,A -85,B 0,C 180,E1 25334.56,E2 25334.56} C_VEL
LIN {X 0,Y 596.757,Z 570.158,A -85,B 0,C 180,E1 25331.483,E2 25331.483} C_VEL
LIN {X 0,Y 595.678,Z 610.202,A -85,B 0,C 180,E1 25330.931,E2 25330.931} C_VEL
LIN {X 0,Y 594.725,Z 617.9,A -85,B 0,C 180,E1 25330.892,E2 25330.892} C_VEL
LIN {X 0,Y 589.616,Z 638.477,A -85,B 0,C 180,E1 25331.02,E2 25331.02} C_VEL
LIN {X 0,Y 588.877,Z 645.081,A -85,B 0,C 180,E1 25330.98,E2 25330.98} C_VEL
LIN {X 0,Y 586.795,Z 713.623,A -85,B 0,C 180,E1 25330.009,E2 25330.009} C_VEL
LIN {X 0,Y 585.039,Z 741.355,A -85,B 0,C 180,E1 25329.454,E2 25329.454} C_VEL
LIN {X 0,Y 583.188,Z 763.474,A -85,B 0,C 180,E1 25328.859,E2 25328.859} C_VEL
LIN {X 0,Y 580.872,Z 786.983,A -85,B 0,C 180,E1 25328.074,E2 25328.074} C_VEL
LIN {X 0,Y 578.028,Z 811.113,A -85,B 0,C 180,E1 25327.074,E2 25327.074} C_VEL
LIN {X 0,Y 575.354,Z 831.253,A -85,B 0,C 180,E1 25326.088,E2 25326.088} C_VEL
LIN {X 0,Y 572.358,Z 852.255,A -85,B 0,C 180,E1 25324.899,E2 25324.899} C_VEL
LIN {X 0,Y 568.795,Z 875.121,A -85,B 0,C 180,E1 25323.382,E2 25323.382} C_VEL
LIN {X 0,Y 565.83,Z 893.077,A -85,B 0,C 180,E1 25322.014,E2 25322.014} C_VEL
LIN {X 0,Y 562.856,Z 910.683,A -85,B 0,C 180,E1 25320.505,E2 25320.505} C_VEL
LIN {X 0,Y 559.141,Z 932.097,A -85,B 0,C 180,E1 25318.403,E2 25318.403} C_VEL
LIN {X 0,Y 556.377,Z 948.281,A -85,B 0,C 180,E1 25316.582,E2 25316.582} C_VEL
LIN {X 0,Y 553.586,Z 965.288,A -85,B 0,C 180,E1 25314.432,E2 25314.432} C_VEL
LIN {X 0,Y 551.075,Z 980.756,A -85,B 0,C 180,E1 25312.173,E2 25312.173} C_VEL
LIN {X 0,Y 549.253,Z 993.181,A -85,B 0,C 180,E1 25310.125,E2 25310.125} C_VEL
LIN {X 0,Y 547.495,Z 1006.456,A -85,B 0,C 180,E1 25307.648,E2 25307.648} C_VEL
LIN {X 0,Y 546.164,Z 1017.73,A -85,B 0,C 180,E1 25305.177,E2 25305.177} C_VEL
LIN {X 0,Y 545.328,Z 1026.259,A -85,B 0,C 180,E1 25303.034,E2 25303.034} C_VEL
LIN {X 0,Y 544.672,Z 1035.013,A -85,B 0,C 180,E1 25300.471,E2 25300.471} C_VEL
LIN {X 0,Y 544.238,Z 1042.248,A -85,B 0,C 180,E1 25297.814,E2 25297.814} C_VEL
LIN {X 0,Y 544.033,Z 1047.099,A -85,B 0,C 180,E1 25295.59,E2 25295.59} C_VEL
LIN {X 0,Y 543.953,Z 1050.836,A -85,B 0,C 180,E1 25293.372,E2 25293.372} C_VEL
LIN {X 0,Y 543.919,Z 1053.967,A -85,B 0,C 180,E1 25290.632,E2 25290.632} C_VEL
LIN {X 0,Y 543.906,Z 1055.237,A -85,B 0,C 180,E1 25288.209,E2 25288.209} C_VEL
LIN {X 0,Y 543.906,Z 1055.3,A -85,B 0,C 180,E1 25285.994,E2 25285.994} C_VEL
LIN {X 0,Y 543.914,Z 1054.287,A -85,B 0,C 180,E1 25283.773,E2 25283.773} C_VEL
LIN {X 0,Y 543.926,Z 1051.709,A -85,B 0,C 180,E1 25281.117,E2 25281.117} C_VEL
LIN {X 0,Y 544.025,Z 1047.547,A -85,B 0,C 180,E1 25278.551,E2 25278.551} C_VEL
LIN {X 0,Y 544.216,Z 1042.709,A -85,B 0,C 180,E1 25276.29,E2 25276.29} C_VEL
LIN {X 0,Y 544.563,Z 1036.364,A -85,B 0,C 180,E1 25273.904,E2 25273.904} C_VEL
LIN {X 0,Y 545.248,Z 1027.212,A -85,B 0,C 180,E1 25271.131,E2 25271.131} C_VEL
LIN {X 0,Y 546.113,Z 1018.249,A -85,B 0,C 180,E1 25268.857,E2 25268.857} C_VEL
LIN {X 0,Y 547.351,Z 1007.557,A -85,B 0,C 180,E1 25266.498,E2 25266.498} C_VEL
LIN {X 0,Y 549.102,Z 994.244,A -85,B 0,C 180,E1 25263.97,E2 25263.97} C_VEL
LIN {X 0,Y 550.935,Z 981.731,A -85,B 0,C 180,E1 25261.89,E2 25261.89} C_VEL
LIN {X 0,Y 553.274,Z 967.041,A -85,B 0,C 180,E1 25259.721,E2 25259.721} C_VEL
LIN {X 0,Y 556.177,Z 949.543,A -85,B 0,C 180,E1 25257.476,E2 25257.476} C_VEL
LIN {X 0,Y 558.844,Z 933.852,A -85,B 0,C 180,E1 25255.695,E2 25255.695} C_VEL
LIN {X 0,Y 562.226,Z 914.537,A -85,B 0,C 180,E1 25253.748,E2 25253.748} C_VEL
LIN {X 0,Y 565.628,Z 894.361,A -85,B 0,C 180,E1 25251.997,E2 25251.997} C_VEL
LIN {X 0,Y 568.478,Z 877.224,A -85,B 0,C 180,E1 25250.675,E2 25250.675} C_VEL
LIN {X 0,Y 571.998,Z 855.483,A -85,B 0,C 180,E1 25249.193,E2 25249.193} C_VEL
LIN {X 0,Y 575.331,Z 832.54,A -85,B 0,C 180,E1 25247.868,E2 25247.868} C_VEL
LIN {X 0,Y 578.037,Z 812.784,A -85,B 0,C 180,E1 25246.885,E2 25246.885} C_VEL
LIN {X 0,Y 580.919,Z 789.573,A -85,B 0,C 180,E1 25245.896,E2 25245.896} C_VEL
LIN {X 0,Y 583.487,Z 764.416,A -85,B 0,C 180,E1 25245.036,E2 25245.036} C_VEL
LIN {X 0,Y 585.375,Z 742.669,A -85,B 0,C 180,E1 25244.44,E2 25244.44} C_VEL
LIN {X 0,Y 587.16,Z 716.836,A -85,B 0,C 180,E1 25243.899,E2 25243.899} C_VEL
LIN {X 0,Y 588.826,Z 668.274,A -85,B 0,C 180,E1 25243.192,E2 25243.192} C_VEL
LIN {X 0,Y 595.678,Z 443.999,A -85,B 0,C 180,E1 25240.021,E2 25240.021} C_VEL
LIN {X 0,Y 598.495,Z 353.222,A -85,B 0,C 180,E1 25238.707,E2 25238.707} C_VEL
LIN {X 0,Y 586.544,Z 334.375,A -85,B 0,C 180,E1 25236.966,E2 25236.966} C_VEL
LIN {X 0,Y 574.086,Z 316.462,A -85,B 0,C 180,E1 25235.022,E2 25235.022} C_VEL
LIN {X 0,Y 564.791,Z 303.865,A -85,B 0,C 180,E1 25233.468,E2 25233.468} C_VEL
LIN {X 0,Y 560.638,Z 298.435,A -85,B 0,C 180,E1 25232.741,E2 25232.741} C_VEL
LIN {X 0,Y 553.15,Z 288.898,A -85,B 0,C 180,E1 25231.373,E2 25231.373} C_VEL
LIN {X 0,Y 548.728,Z 283.465,A -85,B 0,C 180,E1 25230.527,E2 25230.527} C_VEL
LIN {X 0,Y 546.319,Z 280.53,A -85,B 0,C 180,E1 25230.038,E2 25230.038} C_VEL
LIN {X 0,Y 545.573,Z 278.389,A -85,B 0,C 180,E1 25229.659,E2 25229.659} C_VEL
LIN {X 0,Y 545.51,Z 278.024,A -85,B 0,C 180,E1 25228.701,E2 25228.701} C_VEL
LIN {X 0,Y 545.49,Z 277.969,A -85,B 0,C 180,E1 25225.283,E2 25225.283} C_VEL
LIN {X 0,Y 545.566,Z 277.999,A -85,B 0,C 180,E1 25222.069,E2 25222.069} C_VEL
LIN {X 0,Y 545.491,Z 277.978,A -85,B 0,C 180,E1 25218.821,E2 25218.821} C_VEL
LIN {X 0,Y 545.522,Z 277.991,A -85,B 0,C 180,E1 25215.522,E2 25215.522} C_VEL
LIN {X 0,Y 545.499,Z 277.973,A -85,B 0,C 180,E1 25212.491,E2 25212.491} C_VEL
LIN {X 0,Y 545.496,Z 277.998,A -85,B 0,C 180,E1 25209.07,E2 25209.07} C_VEL
LIN {X 0,Y 545.547,Z 277.957,A -85,B 0,C 180,E1 25205.891,E2 25205.891} C_VEL
LIN {X 0,Y 545.494,Z 278.017,A -85,B 0,C 180,E1 25202.627,E2 25202.627} C_VEL
LIN {X 0,Y 545.532,Z 277.955,A -85,B 0,C 180,E1 25199.37,E2 25199.37} C_VEL
LIN {X 0,Y 545.507,Z 278.032,A -85,B 0,C 180,E1 25196.216,E2 25196.216} C_VEL
LIN {X 0,Y 545.494,Z 277.952,A -85,B 0,C 180,E1 25192.84,E2 25192.84} C_VEL
LIN {X 0,Y 545.549,Z 278.023,A -85,B 0,C 180,E1 25189.653,E2 25189.653} C_VEL
LIN {X 0,Y 545.486,Z 277.955,A -85,B 0,C 180,E1 25186.43,E2 25186.43} C_VEL
LIN {X 0,Y 545.547,Z 278.022,A -85,B 0,C 180,E1 25183.167,E2 25183.167} C_VEL
LIN {X 0,Y 545.5,Z 277.96,A -85,B 0,C 180,E1 25179.954,E2 25179.954} C_VEL
LIN {X 0,Y 545.504,Z 278.032,A -85,B 0,C 180,E1 25176.562,E2 25176.562} C_VEL
LIN {X 0,Y 545.557,Z 278.027,A -85,B 0,C 180,E1 25173.318,E2 25173.318} C_VEL
LIN {X 0,Y 545.498,Z 278.034,A -85,B 0,C 180,E1 25170.094,E2 25170.094} C_VEL
LIN {X 0,Y 545.529,Z 278.255,A -85,B 0,C 180,E1 25168.117,E2 25168.117} C_VEL
LIN {X 0,Y 546.932,Z 281.564,A -85,B 0,C 180,E1 25167.363,E2 25167.363} C_VEL
LIN {X 0,Y 548.166,Z 283.805,A -85,B 0,C 180,E1 25166.85,E2 25166.85} C_VEL
LIN {X 0,Y 549.497,Z 286.328,A -85,B 0,C 180,E1 25166.384,E2 25166.384} C_VEL
LIN {X 0,Y 555.721,Z 294.251,A -85,B 0,C 180,E1 25165.193,E2 25165.193} C_VEL
LIN {X 0,Y 564.194,Z 305.393,A -85,B 0,C 180,E1 25163.674,E2 25163.674} C_VEL
LIN {X 0,Y 574.04,Z 319.019,A -85,B 0,C 180,E1 25162.025,E2 25162.025} C_VEL
LIN {X 0,Y 585.961,Z 336.353,A -85,B 0,C 180,E1 25160.164,E2 25160.164} C_VEL
LIN {X 0,Y 597.599,Z 354.907,A -85,B 0,C 180,E1 25158.455,E2 25158.455} C_VEL
LIN {X 0,Y 598.666,Z 357.042,A -85,B 0,C 180,E1 25158.297,E2 25158.297} C_VEL
LIN {X 0,Y 591.378,Z 587.212,A -85,B 0,C 180,E1 25155.027,E2 25155.027} C_VEL
LIN {X 0,Y 587.269,Z 720.394,A -85,B 0,C 180,E1 25153.14,E2 25153.14} C_VEL
LIN {X 0,Y 585.543,Z 747.441,A -85,B 0,C 180,E1 25152.615,E2 25152.615} C_VEL
LIN {X 0,Y 583.52,Z 770.841,A -85,B 0,C 180,E1 25151.992,E2 25151.992} C_VEL
LIN {X 0,Y 581.262,Z 792.991,A -85,B 0,C 180,E1 25151.259,E2 25151.259} C_VEL
LIN {X 0,Y 578.093,Z 819.415,A -85,B 0,C 180,E1 25150.177,E2 25150.177} C_VEL
LIN {X 0,Y 575.351,Z 839.617,A -85,B 0,C 180,E1 25149.186,E2 25149.186} C_VEL
LIN {X 0,Y 572.333,Z 860.414,A -85,B 0,C 180,E1 25148.008,E2 25148.008} C_VEL
LIN {X 0,Y 568.678,Z 883.794,A -85,B 0,C 180,E1 25146.462,E2 25146.462} C_VEL
LIN {X 0,Y 565.65,Z 902.184,A -85,B 0,C 180,E1 25145.064,E2 25145.064} C_VEL
LIN {X 0,Y 562.684,Z 919.937,A -85,B 0,C 180,E1 25143.549,E2 25143.549} C_VEL
LIN {X 0,Y 558.976,Z 941.598,A -85,B 0,C 180,E1 25141.432,E2 25141.432} C_VEL
LIN {X 0,Y 556.337,Z 957.299,A -85,B 0,C 180,E1 25139.679,E2 25139.679} C_VEL
LIN {X 0,Y 553.714,Z 973.529,A -85,B 0,C 180,E1 25137.651,E2 25137.651} C_VEL
LIN {X 0,Y 551.159,Z 989.622,A -85,B 0,C 180,E1 25135.35,E2 25135.35} C_VEL
LIN {X 0,Y 549.305,Z 1002.446,A -85,B 0,C 180,E1 25133.266,E2 25133.266} C_VEL
LIN {X 0,Y 547.585,Z 1015.566,A -85,B 0,C 180,E1 25130.859,E2 25130.859} C_VEL
LIN {X 0,Y 546.224,Z 1027.176,A -85,B 0,C 180,E1 25128.352,E2 25128.352} C_VEL
LIN {X 0,Y 545.368,Z 1035.875,A -85,B 0,C 180,E1 25126.181,E2 25126.181} C_VEL
LIN {X 0,Y 544.739,Z 1043.983,A -85,B 0,C 180,E1 25123.831,E2 25123.831} C_VEL
LIN {X 0,Y 544.25,Z 1051.877,A -85,B 0,C 180,E1 25121.015,E2 25121.015} C_VEL
LIN {X 0,Y 544.039,Z 1056.828,A -85,B 0,C 180,E1 25118.774,E2 25118.774} C_VEL
LIN {X 0,Y 543.961,Z 1060.486,A -85,B 0,C 180,E1 25116.65,E2 25116.65} C_VEL
LIN {X 0,Y 543.911,Z 1063.469,A -85,B 0,C 180,E1 25114.217,E2 25114.217} C_VEL
LIN {X 0,Y 543.898,Z 1065.19,A -85,B 0,C 180,E1 25111.475,E2 25111.475} C_VEL
LIN {X 0,Y 543.899,Z 1065.348,A -85,B 0,C 180,E1 25109.263,E2 25109.263} C_VEL
LIN {X 0,Y 543.913,Z 1064.436,A -85,B 0,C 180,E1 25107.05,E2 25107.05} C_VEL
LIN {X 0,Y 543.922,Z 1062.446,A -85,B 0,C 180,E1 25104.832,E2 25104.832} C_VEL
LIN {X 0,Y 544.014,Z 1058.48,A -85,B 0,C 180,E1 25102.077,E2 25102.077} C_VEL
LIN {X 0,Y 544.177,Z 1053.403,A -85,B 0,C 180,E1 25099.626,E2 25099.626} C_VEL
LIN {X 0,Y 544.465,Z 1047.875,A -85,B 0,C 180,E1 25097.485,E2 25097.485} C_VEL
LIN {X 0,Y 544.958,Z 1040.886,A -85,B 0,C 180,E1 25095.224,E2 25095.224} C_VEL
LIN {X 0,Y 545.896,Z 1030.391,A -85,B 0,C 180,E1 25092.409,E2 25092.409} C_VEL
LIN {X 0,Y 546.935,Z 1020.804,A -85,B 0,C 180,E1 25090.232,E2 25090.232} C_VEL
LIN {X 0,Y 548.239,Z 1010.387,A -85,B 0,C 180,E1 25088.158,E2 25088.158} C_VEL
LIN {X 0,Y 550.243,Z 995.965,A -85,B 0,C 180,E1 25085.638,E2 25085.638} C_VEL
LIN {X 0,Y 552.422,Z 981.427,A -85,B 0,C 180,E1 25083.444,E2 25083.444} C_VEL
LIN {X 0,Y 554.639,Z 967.597,A -85,B 0,C 180,E1 25081.58,E2 25081.58} C_VEL
LIN {X 0,Y 557.757,Z 949.097,A -85,B 0,C 180,E1 25079.373,E2 25079.373} C_VEL
LIN {X 0,Y 560.718,Z 931.448,A -85,B 0,C 180,E1 25077.537,E2 25077.537} C_VEL
LIN {X 0,Y 563.628,Z 914.236,A -85,B 0,C 180,E1 25075.942,E2 25075.942} C_VEL
LIN {X 0,Y 567.375,Z 891.711,A -85,B 0,C 180,E1 25074.116,E2 25074.116} C_VEL
LIN {X 0,Y 570.375,Z 872.744,A -85,B 0,C 180,E1 25072.786,E2 25072.786} C_VEL
LIN {X 0,Y 573.232,Z 853.775,A -85,B 0,C 180,E1 25071.613,E2 25071.613} C_VEL
LIN {X 0,Y 576.584,Z 830.015,A -85,B 0,C 180,E1 25070.345,E2 25070.345} C_VEL
LIN {X 0,Y 579.352,Z 807.529,A -85,B 0,C 180,E1 25069.344,E2 25069.344} C_VEL
LIN {X 0,Y 581.481,Z 788.191,A -85,B 0,C 180,E1 25068.611,E2 25068.611} C_VEL
LIN {X 0,Y 583.693,Z 765.447,A -85,B 0,C 180,E1 25067.895,E2 25067.895} C_VEL
LIN {X 0,Y 585.699,Z 739.383,A -85,B 0,C 180,E1 25067.263,E2 25067.263} C_VEL
LIN {X 0,Y 586.911,Z 717.15,A -85,B 0,C 180,E1 25066.863,E2 25066.863} C_VEL
LIN {X 0,Y 593.472,Z 487.752,A -85,B 0,C 180,E1 25063.66,E2 25063.66} C_VEL
LIN {X 0,Y 597.277,Z 356.318,A -85,B 0,C 180,E1 25061.798,E2 25061.798} C_VEL
LIN {X 0,Y 582.016,Z 332.467,A -85,B 0,C 180,E1 25059.724,E2 25059.724} C_VEL
LIN {X 0,Y 570.727,Z 315.728,A -85,B 0,C 180,E1 25058.075,E2 25058.075} C_VEL
LIN {X 0,Y 560.589,Z 301.451,A -85,B 0,C 180,E1 25056.502,E2 25056.502} C_VEL
LIN {X 0,Y 552.977,Z 291.223,A -85,B 0,C 180,E1 25055.259,E2 25055.259} C_VEL
LIN {X 0,Y 549.048,Z 285.81,A -85,B 0,C 180,E1 25054.561,E2 25054.561} C_VEL
LIN {X 0,Y 546.933,Z 281.65,A -85,B 0,C 180,E1 25053.764,E2 25053.764} C_VEL
LIN {X 0,Y 545.576,Z 278.191,A -85,B 0,C 180,E1 25053.055,E2 25053.055} C_VEL
LIN {X 0,Y 545.492,Z 277.979,A -85,B 0,C 180,E1 25049.785,E2 25049.785} C_VEL
LIN {X 0,Y 545.542,Z 278.001,A -85,B 0,C 180,E1 25046.565,E2 25046.565} C_VEL
LIN {X 0,Y 545.502,Z 278.012,A -85,B 0,C 180,E1 25043.438,E2 25043.438} C_VEL
LIN {X 0,Y 545.506,Z 278.01,A -85,B 0,C 180,E1 25040.045,E2 25040.045} C_VEL
LIN {X 0,Y 545.544,Z 278.006,A -85,B 0,C 180,E1 25036.833,E2 25036.833} C_VEL
LIN {X 0,Y 545.495,Z 278.024,A -85,B 0,C 180,E1 25033.678,E2 25033.678} C_VEL
LIN {X 0,Y 545.556,Z 278.027,A -85,B 0,C 180,E1 25030.454,E2 25030.454} C_VEL
LIN {X 0,Y 545.495,Z 278.021,A -85,B 0,C 180,E1 25027.266,E2 25027.266} C_VEL
LIN {X 0,Y 545.512,Z 278.007,A -85,B 0,C 180,E1 25023.889,E2 25023.889} C_VEL
LIN {X 0,Y 545.528,Z 278.012,A -85,B 0,C 180,E1 25020.735,E2 25020.735} C_VEL
LIN {X 0,Y 545.495,Z 278.03,A -85,B 0,C 180,E1 25017.405,E2 25017.405} C_VEL
LIN {X 0,Y 545.554,Z 278.016,A -85,B 0,C 180,E1 25014.109,E2 25014.109} C_VEL
LIN {X 0,Y 545.498,Z 278.006,A -85,B 0,C 180,E1 25010.93,E2 25010.93} C_VEL
LIN {X 0,Y 545.503,Z 278.006,A -85,B 0,C 180,E1 25007.509,E2 25007.509} C_VEL
LIN {X 0,Y 545.539,Z 278.021,A -85,B 0,C 180,E1 25004.37,E2 25004.37} C_VEL
LIN {X 0,Y 545.496,Z 278.031,A -85,B 0,C 180,E1 25001.053,E2 25001.053} C_VEL
LIN {X 0,Y 545.544,Z 278.018,A -85,B 0,C 180,E1 24997.755,E2 24997.755} C_VEL
LIN {X 0,Y 545.493,Z 277.954,A -85,B 0,C 180,E1 24994.601,E2 24994.601} C_VEL
LIN {X 0,Y 545.498,Z 277.998,A -85,B 0,C 180,E1 24991.179,E2 24991.179} C_VEL
LIN {X 0,Y 545.515,Z 277.965,A -85,B 0,C 180,E1 24988.261,E2 24988.261} C_VEL
LIN {X 0,Y 545.493,Z 277.984,A -85,B 0,C 180,E1 24984.989,E2 24984.989} C_VEL
LIN {X 0,Y 545.544,Z 278.297,A -85,B 0,C 180,E1 24983.122,E2 24983.122} C_VEL
LIN {X 0,Y 546.213,Z 280.473,A -85,B 0,C 180,E1 24982.778,E2 24982.778} C_VEL
LIN {X 0,Y 548.543,Z 283.342,A -85,B 0,C 180,E1 24982.364,E2 24982.364} C_VEL
LIN {X 0,Y 554.594,Z 291.139,A -85,B 0,C 180,E1 24981.339,E2 24981.339} C_VEL
LIN {X 0,Y 561.394,Z 300.166,A -85,B 0,C 180,E1 24980.235,E2 24980.235} C_VEL
LIN {X 0,Y 572.192,Z 315.198,A -85,B 0,C 180,E1 24978.575,E2 24978.575} C_VEL
LIN {X 0,Y 586.316,Z 336.04,A -85,B 0,C 180,E1 24976.552,E2 24976.552} C_VEL
LIN {X 0,Y 597.299,Z 353.39,A -85,B 0,C 180,E1 24975.069,E2 24975.069} C_VEL
LIN {X 0,Y 590.934,Z 571.693,A -85,B 0,C 180,E1 24971.999,E2 24971.999} C_VEL
LIN {X 0,Y 588.877,Z 645.081,A -85,B 0,C 180,E1 24970.98,E2 24970.98} C_VEL
LIN {X 0,Y 587.921,Z 652.781,A -85,B 0,C 180,E1 24970.941,E2 24970.941} C_VEL
LIN {X 0,Y 582.777,Z 673.354,A -85,B 0,C 180,E1 24971.074,E2 24971.074} C_VEL
LIN {X 0,Y 582.048,Z 679.958,A -85,B 0,C 180,E1 24971.032,E2 24971.032} C_VEL
LIN {X 0,Y 580.621,Z 719.149,A -85,B 0,C 180,E1 24970.449,E2 24970.449} C_VEL
LIN {X 0,Y 578.885,Z 743.596,A -85,B 0,C 180,E1 24969.928,E2 24969.928} C_VEL
LIN {X 0,Y 576.975,Z 765.347,A -85,B 0,C 180,E1 24969.33,E2 24969.33} C_VEL
LIN {X 0,Y 574.268,Z 791.254,A -85,B 0,C 180,E1 24968.432,E2 24968.432} C_VEL
LIN {X 0,Y 571.534,Z 813.015,A -85,B 0,C 180,E1 24967.504,E2 24967.504} C_VEL
LIN {X 0,Y 568.785,Z 832.848,A -85,B 0,C 180,E1 24966.517,E2 24966.517} C_VEL
LIN {X 0,Y 565.418,Z 855.556,A -85,B 0,C 180,E1 24965.205,E2 24965.205} C_VEL
LIN {X 0,Y 561.955,Z 876.453,A -85,B 0,C 180,E1 24963.782,E2 24963.782} C_VEL
LIN {X 0,Y 558.994,Z 893.681,A -85,B 0,C 180,E1 24962.453,E2 24962.453} C_VEL
LIN {X 0,Y 555.834,Z 911.609,A -85,B 0,C 180,E1 24960.898,E2 24960.898} C_VEL
LIN {X 0,Y 551.999,Z 932.609,A -85,B 0,C 180,E1 24958.805,E2 24958.805} C_VEL
LIN {X 0,Y 549.252,Z 947.852,A -85,B 0,C 180,E1 24957.072,E2 24957.072} C_VEL
LIN {X 0,Y 546.546,Z 963.38,A -85,B 0,C 180,E1 24955.097,E2 24955.097} C_VEL
LIN {X 0,Y 543.746,Z 979.765,A -85,B 0,C 180,E1 24952.716,E2 24952.716} C_VEL
LIN {X 0,Y 541.772,Z 992.289,A -85,B 0,C 180,E1 24950.641,E2 24950.641} C_VEL
LIN {X 0,Y 540.084,Z 1003.998,A -85,B 0,C 180,E1 24948.456,E2 24948.456} C_VEL
LIN {X 0,Y 538.474,Z 1016.611,A -85,B 0,C 180,E1 24945.73,E2 24945.73} C_VEL
LIN {X 0,Y 537.47,Z 1026.032,A -85,B 0,C 180,E1 24943.337,E2 24943.337} C_VEL
LIN {X 0,Y 536.773,Z 1034.465,A -85,B 0,C 180,E1 24940.844,E2 24940.844} C_VEL
LIN {X 0,Y 536.269,Z 1042.007,A -85,B 0,C 180,E1 24938.08,E2 24938.08} C_VEL
LIN {X 0,Y 536.046,Z 1046.982,A -85,B 0,C 180,E1 24935.781,E2 24935.781} C_VEL
LIN {X 0,Y 535.958,Z 1050.753,A -85,B 0,C 180,E1 24933.524,E2 24933.524} C_VEL
LIN {X 0,Y 535.921,Z 1053.927,A -85,B 0,C 180,E1 24930.748,E2 24930.748} C_VEL
LIN {X 0,Y 535.907,Z 1055.246,A -85,B 0,C 180,E1 24928.182,E2 24928.182} C_VEL
LIN {X 0,Y 535.907,Z 1055.291,A -85,B 0,C 180,E1 24925.934,E2 24925.934} C_VEL
LIN {X 0,Y 535.912,Z 1054.258,A -85,B 0,C 180,E1 24923.68,E2 24923.68} C_VEL
LIN {X 0,Y 535.935,Z 1051.641,A -85,B 0,C 180,E1 24920.984,E2 24920.984} C_VEL
LIN {X 0,Y 536.035,Z 1047.458,A -85,B 0,C 180,E1 24918.378,E2 24918.378} C_VEL
LIN {X 0,Y 536.233,Z 1042.855,A -85,B 0,C 180,E1 24916.192,E2 24916.192} C_VEL
LIN {X 0,Y 536.581,Z 1036.845,A -85,B 0,C 180,E1 24913.88,E2 24913.88} C_VEL
LIN {X 0,Y 537.286,Z 1028.001,A -85,B 0,C 180,E1 24911.106,E2 24911.106} C_VEL
LIN {X 0,Y 538.25,Z 1018.54,A -85,B 0,C 180,E1 24908.648,E2 24908.648} C_VEL
LIN {X 0,Y 539.553,Z 1008.018,A -85,B 0,C 180,E1 24906.274,E2 24906.274} C_VEL
LIN {X 0,Y 541.524,Z 994.035,A -85,B 0,C 180,E1 24903.576,E2 24903.576} C_VEL
LIN {X 0,Y 543.391,Z 981.931,A -85,B 0,C 180,E1 24901.538,E2 24901.538} C_VEL
LIN {X 0,Y 545.825,Z 967.558,A -85,B 0,C 180,E1 24899.385,E2 24899.385} C_VEL
LIN {X 0,Y 548.934,Z 949.736,A -85,B 0,C 180,E1 24897.063,E2 24897.063} C_VEL
LIN {X 0,Y 551.752,Z 933.992,A -85,B 0,C 180,E1 24895.254,E2 24895.254} C_VEL
LIN {X 0,Y 555.321,Z 914.698,A -85,B 0,C 180,E1 24893.289,E2 24893.289} C_VEL
LIN {X 0,Y 558.79,Z 895.146,A -85,B 0,C 180,E1 24891.566,E2 24891.566} C_VEL
LIN {X 0,Y 561.79,Z 878.007,A -85,B 0,C 180,E1 24890.225,E2 24890.225} C_VEL
LIN {X 0,Y 565.009,Z 858.963,A -85,B 0,C 180,E1 24888.902,E2 24888.902} C_VEL
LIN {X 0,Y 568.844,Z 834.348,A -85,B 0,C 180,E1 24887.435,E2 24887.435} C_VEL
LIN {X 0,Y 571.666,Z 814.697,A -85,B 0,C 180,E1 24886.438,E2 24886.438} C_VEL
LIN {X 0,Y 574.34,Z 794.206,A -85,B 0,C 180,E1 24885.544,E2 24885.544} C_VEL
LIN {X 0,Y 577.201,Z 768.904,A -85,B 0,C 180,E1 24884.629,E2 24884.629} C_VEL
LIN {X 0,Y 579.327,Z 745.722,A -85,B 0,C 180,E1 24883.969,E2 24883.969} C_VEL
LIN {X 0,Y 580.901,Z 724.894,A -85,B 0,C 180,E1 24883.505,E2 24883.505} C_VEL
LIN {X 0,Y 582.244,Z 698.099,A -85,B 0,C 180,E1 24883.056,E2 24883.056} C_VEL
LIN {X 0,Y 589.767,Z 461.933,A -85,B 0,C 180,E1 24879.701,E2 24879.701} C_VEL
LIN {X 0,Y 593.164,Z 356.986,A -85,B 0,C 180,E1 24878.172,E2 24878.172} C_VEL
LIN {X 0,Y 581.861,Z 339.19,A -85,B 0,C 180,E1 24876.483,E2 24876.483} C_VEL
LIN {X 0,Y 569.193,Z 320.77,A -85,B 0,C 180,E1 24874.448,E2 24874.448} C_VEL
LIN {X 0,Y 557.671,Z 305.296,A -85,B 0,C 180,E1 24872.449,E2 24872.449} C_VEL
LIN {X 0,Y 549.886,Z 295.39,A -85,B 0,C 180,E1 24871.001,E2 24871.001} C_VEL
LIN {X 0,Y 545.867,Z 290.402,A -85,B 0,C 180,E1 24870.217,E2 24870.217} C_VEL
LIN {X 0,Y 542.982,Z 286.698,A -85,B 0,C 180,E1 24869.633,E2 24869.633} C_VEL
LIN {X 0,Y 541.605,Z 285.028,A -85,B 0,C 180,E1 24869.351,E2 24869.351} C_VEL
LIN {X 0,Y 538.924,Z 282.573,A -85,B 0,C 180,E1 24868.811,E2 24868.811} C_VEL
LIN {X 0,Y 537.683,Z 279.543,A -85,B 0,C 180,E1 24868.406,E2 24868.406} C_VEL
LIN {X 0,Y 537.596,Z 278.991,A -85,B 0,C 180,E1 24867.83,E2 24867.83} C_VEL
LIN {X 0,Y 537.57,Z 278.966,A -85,B 0,C 180,E1 24864.558,E2 24864.558} C_VEL
LIN {X 0,Y 537.558,Z 278.966,A -85,B 0,C 180,E1 24861.267,E2 24861.267} C_VEL
LIN {X 0,Y 537.618,Z 278.982,A -85,B 0,C 180,E1 24857.983,E2 24857.983} C_VEL
LIN {X 0,Y 537.551,Z 278.958,A -85,B 0,C 180,E1 24854.764,E2 24854.764} C_VEL
LIN {X 0,Y 537.578,Z 278.994,A -85,B 0,C 180,E1 24851.371,E2 24851.371} C_VEL
LIN {X 0,Y 537.574,Z 278.953,A -85,B 0,C 180,E1 24848.234,E2 24848.234} C_VEL
LIN {X 0,Y 537.555,Z 278.981,A -85,B 0,C 180,E1 24844.908,E2 24844.908} C_VEL
LIN {X 0,Y 537.616,Z 278.962,A -85,B 0,C 180,E1 24841.705,E2 24841.705} C_VEL
LIN {X 0,Y 537.552,Z 278.965,A -85,B 0,C 180,E1 24838.508,E2 24838.508} C_VEL
LIN {X 0,Y 537.585,Z 278.986,A -85,B 0,C 180,E1 24835.199,E2 24835.199} C_VEL
LIN {X 0,Y 537.564,Z 278.945,A -85,B 0,C 180,E1 24832.088,E2 24832.088} C_VEL
LIN {X 0,Y 537.561,Z 279.002,A -85,B 0,C 180,E1 24828.737,E2 24828.737} C_VEL
LIN {X 0,Y 537.62,Z 278.936,A -85,B 0,C 180,E1 24825.459,E2 24825.459} C_VEL
LIN {X 0,Y 537.558,Z 279.006,A -85,B 0,C 180,E1 24822.239,E2 24822.239} C_VEL
LIN {X 0,Y 537.575,Z 278.951,A -85,B 0,C 180,E1 24818.848,E2 24818.848} C_VEL
LIN {X 0,Y 537.571,Z 279.007,A -85,B 0,C 180,E1 24815.845,E2 24815.845} C_VEL
LIN {X 0,Y 537.563,Z 279.006,A -85,B 0,C 180,E1 24812.409,E2 24812.409} C_VEL
LIN {X 0,Y 537.634,Z 279.218,A -85,B 0,C 180,E1 24809.403,E2 24809.403} C_VEL
LIN {X 0,Y 539.327,Z 283.07,A -85,B 0,C 180,E1 24808.478,E2 24808.478} C_VEL
LIN {X 0,Y 540.888,Z 286.022,A -85,B 0,C 180,E1 24807.863,E2 24807.863} C_VEL
LIN {X 0,Y 545.447,Z 291.742,A -85,B 0,C 180,E1 24806.919,E2 24806.919} C_VEL
LIN {X 0,Y 552.698,Z 301.025,A -85,B 0,C 180,E1 24805.511,E2 24805.511} C_VEL
LIN {X 0,Y 561.334,Z 312.526,A -85,B 0,C 180,E1 24803.934,E2 24803.934} C_VEL
LIN {X 0,Y 570.514,Z 325.333,A -85,B 0,C 180,E1 24802.369,E2 24802.369} C_VEL
LIN {X 0,Y 582.174,Z 342.444,A -85,B 0,C 180,E1 24800.512,E2 24800.512} C_VEL
LIN {X 0,Y 593.338,Z 360.411,A -85,B 0,C 180,E1 24798.838,E2 24798.838} C_VEL
LIN {X 0,Y 585.855,Z 586.302,A -85,B 0,C 180,E1 24795.604,E2 24795.604} C_VEL
LIN {X 0,Y 581.528,Z 720.248,A -85,B 0,C 180,E1 24793.691,E2 24793.691} C_VEL
LIN {X 0,Y 579.745,Z 747.26,A -85,B 0,C 180,E1 24793.165,E2 24793.165} C_VEL
LIN {X 0,Y 577.629,Z 770.762,A -85,B 0,C 180,E1 24792.537,E2 24792.537} C_VEL
LIN {X 0,Y 575.282,Z 792.879,A -85,B 0,C 180,E1 24791.801,E2 24791.801} C_VEL
LIN {X 0,Y 571.925,Z 819.593,A -85,B 0,C 180,E1 24790.701,E2 24790.701} C_VEL
LIN {X 0,Y 568.977,Z 840.369,A -85,B 0,C 180,E1 24789.671,E2 24789.671} C_VEL
LIN {X 0,Y 565.529,Z 863.145,A -85,B 0,C 180,E1 24788.359,E2 24788.359} C_VEL
LIN {X 0,Y 561.827,Z 885.29,A -85,B 0,C 180,E1 24786.853,E2 24786.853} C_VEL
LIN {X 0,Y 558.782,Z 902.874,A -85,B 0,C 180,E1 24785.493,E2 24785.493} C_VEL
LIN {X 0,Y 555.318,Z 922.641,A -85,B 0,C 180,E1 24783.771,E2 24783.771} C_VEL
LIN {X 0,Y 551.735,Z 942.342,A -85,B 0,C 180,E1 24781.793,E2 24781.793} C_VEL
LIN {X 0,Y 549.021,Z 957.677,A -85,B 0,C 180,E1 24780.055,E2 24780.055} C_VEL
LIN {X 0,Y 546.202,Z 974.292,A -85,B 0,C 180,E1 24777.946,E2 24777.946} C_VEL
LIN {X 0,Y 543.519,Z 990.241,A -85,B 0,C 180,E1 24775.615,E2 24775.615} C_VEL
LIN {X 0,Y 541.573,Z 1003,A -85,B 0,C 180,E1 24773.503,E2 24773.503} C_VEL
LIN {X 0,Y 539.697,Z 1016.58,A -85,B 0,C 180,E1 24770.951,E2 24770.951} C_VEL
LIN {X 0,Y 538.34,Z 1027.6,A -85,B 0,C 180,E1 24768.518,E2 24768.518} C_VEL
LIN {X 0,Y 537.486,Z 1035.874,A -85,B 0,C 180,E1 24766.425,E2 24766.425} C_VEL
LIN {X 0,Y 536.796,Z 1044.066,A -85,B 0,C 180,E1 24764.013,E2 24764.013} C_VEL
LIN {X 0,Y 536.275,Z 1051.877,A -85,B 0,C 180,E1 24761.181,E2 24761.181} C_VEL
LIN {X 0,Y 536.052,Z 1056.828,A -85,B 0,C 180,E1 24758.906,E2 24758.906} C_VEL
LIN {X 0,Y 535.963,Z 1060.486,A -85,B 0,C 180,E1 24756.75,E2 24756.75} C_VEL
LIN {X 0,Y 535.907,Z 1063.356,A -85,B 0,C 180,E1 24754.387,E2 24754.387} C_VEL
LIN {X 0,Y 535.897,Z 1065.167,A -85,B 0,C 180,E1 24751.604,E2 24751.604} C_VEL
LIN {X 0,Y 535.9,Z 1065.348,A -85,B 0,C 180,E1 24749.252,E2 24749.252} C_VEL
LIN {X 0,Y 535.913,Z 1064.435,A -85,B 0,C 180,E1 24747.005,E2 24747.005} C_VEL
LIN {X 0,Y 535.924,Z 1062.446,A -85,B 0,C 180,E1 24744.755,E2 24744.755} C_VEL
LIN {X 0,Y 536.017,Z 1058.48,A -85,B 0,C 180,E1 24741.958,E2 24741.958} C_VEL
LIN {X 0,Y 536.205,Z 1053.403,A -85,B 0,C 180,E1 24739.47,E2 24739.47} C_VEL
LIN {X 0,Y 536.512,Z 1047.875,A -85,B 0,C 180,E1 24737.296,E2 24737.296} C_VEL
LIN {X 0,Y 537.043,Z 1040.886,A -85,B 0,C 180,E1 24735.002,E2 24735.002} C_VEL
LIN {X 0,Y 538.047,Z 1030.373,A -85,B 0,C 180,E1 24732.144,E2 24732.144} C_VEL
LIN {X 0,Y 539.219,Z 1020.214,A -85,B 0,C 180,E1 24729.824,E2 24729.824} C_VEL
LIN {X 0,Y 540.769,Z 1008.576,A -85,B 0,C 180,E1 24727.496,E2 24727.496} C_VEL
LIN {X 0,Y 542.982,Z 993.772,A -85,B 0,C 180,E1 24724.942,E2 24724.942} C_VEL
LIN {X 0,Y 545.091,Z 980.571,A -85,B 0,C 180,E1 24722.94,E2 24722.94} C_VEL
LIN {X 0,Y 547.631,Z 965.817,A -85,B 0,C 180,E1 24720.944,E2 24720.944} C_VEL
LIN {X 0,Y 550.997,Z 946.657,A -85,B 0,C 180,E1 24718.674,E2 24718.674} C_VEL
LIN {X 0,Y 554.006,Z 929.692,A -85,B 0,C 180,E1 24716.91,E2 24716.91} C_VEL
LIN {X 0,Y 557.533,Z 910.085,A -85,B 0,C 180,E1 24715.103,E2 24715.103} C_VEL
LIN {X 0,Y 561.123,Z 889.009,A -85,B 0,C 180,E1 24713.435,E2 24713.435} C_VEL
LIN {X 0,Y 564.1,Z 870.905,A -85,B 0,C 180,E1 24712.172,E2 24712.172} C_VEL
LIN {X 0,Y 567.395,Z 849.902,A -85,B 0,C 180,E1 24710.885,E2 24710.885} C_VEL
LIN {X 0,Y 570.767,Z 825.998,A -85,B 0,C 180,E1 24709.646,E2 24709.646} C_VEL
LIN {X 0,Y 573.337,Z 805.867,A -85,B 0,C 180,E1 24708.76,E2 24708.76} C_VEL
LIN {X 0,Y 575.57,Z 786.272,A -85,B 0,C 180,E1 24708.024,E2 24708.024} C_VEL
LIN {X 0,Y 578.072,Z 761.04,A -85,B 0,C 180,E1 24707.246,E2 24707.246} C_VEL
LIN {X 0,Y 579.88,Z 737.076,A -85,B 0,C 180,E1 24706.688,E2 24706.688} C_VEL
LIN {X 0,Y 581.064,Z 715.442,A -85,B 0,C 180,E1 24706.306,E2 24706.306} C_VEL
LIN {X 0,Y 588.071,Z 480.499,A -85,B 0,C 180,E1 24703.002,E2 24703.002} C_VEL
LIN {X 0,Y 591.68,Z 359.94,A -85,B 0,C 180,E1 24701.277,E2 24701.277} C_VEL
LIN {X 0,Y 575.832,Z 335.035,A -85,B 0,C 180,E1 24699.058,E2 24699.058} C_VEL
LIN {X 0,Y 562.328,Z 315.151,A -85,B 0,C 180,E1 24697.006,E2 24697.006} C_VEL
LIN {X 0,Y 553.318,Z 302.778,A -85,B 0,C 180,E1 24695.551,E2 24695.551} C_VEL
LIN {X 0,Y 545.377,Z 292.07,A -85,B 0,C 180,E1 24694.19,E2 24694.19} C_VEL
LIN {X 0,Y 540.399,Z 285.419,A -85,B 0,C 180,E1 24693.246,E2 24693.246} C_VEL
LIN {X 0,Y 539.292,Z 282.978,A -85,B 0,C 180,E1 24692.779,E2 24692.779} C_VEL
LIN {X 0,Y 537.61,Z 279.359,A -85,B 0,C 180,E1 24692.01,E2 24692.01} C_VEL
LIN {X 0,Y 537.607,Z 278.986,A -85,B 0,C 180,E1 24690.638,E2 24690.638} C_VEL
LIN {X 0,Y 537.561,Z 278.963,A -85,B 0,C 180,E1 24687.471,E2 24687.471} C_VEL
LIN {X 0,Y 537.563,Z 278.999,A -85,B 0,C 180,E1 24684.038,E2 24684.038} C_VEL
LIN {X 0,Y 537.605,Z 278.997,A -85,B 0,C 180,E1 24680.922,E2 24680.922} C_VEL
LIN {X 0,Y 537.557,Z 279.012,A -85,B 0,C 180,E1 24677.649,E2 24677.649} C_VEL
LIN {X 0,Y 537.601,Z 279.015,A -85,B 0,C 180,E1 24674.322,E2 24674.322} C_VEL
LIN {X 0,Y 537.568,Z 279.014,A -85,B 0,C 180,E1 24671.154,E2 24671.154} C_VEL
LIN {X 0,Y 537.557,Z 279.001,A -85,B 0,C 180,E1 24667.696,E2 24667.696} C_VEL
LIN {X 0,Y 537.614,Z 278.99,A -85,B 0,C 180,E1 24664.48,E2 24664.48} C_VEL
LIN {X 0,Y 537.56,Z 279.013,A -85,B 0,C 180,E1 24661.172,E2 24661.172} C_VEL
LIN {X 0,Y 537.572,Z 279.02,A -85,B 0,C 180,E1 24657.761,E2 24657.761} C_VEL
LIN {X 0,Y 537.607,Z 279,A -85,B 0,C 180,E1 24654.45,E2 24654.45} C_VEL
LIN {X 0,Y 537.553,Z 278.994,A -85,B 0,C 180,E1 24651.227,E2 24651.227} C_VEL
LIN {X 0,Y 537.606,Z 278.996,A -85,B 0,C 180,E1 24647.977,E2 24647.977} C_VEL
LIN {X 0,Y 537.564,Z 279.019,A -85,B 0,C 180,E1 24644.795,E2 24644.795} C_VEL
LIN {X 0,Y 537.565,Z 279.02,A -85,B 0,C 180,E1 24641.341,E2 24641.341} C_VEL
LIN {X 0,Y 537.626,Z 278.998,A -85,B 0,C 180,E1 24638.048,E2 24638.048} C_VEL
LIN {X 0,Y 537.547,Z 278.945,A -85,B 0,C 180,E1 24634.788,E2 24634.788} C_VEL
LIN {X 0,Y 537.572,Z 278.971,A -85,B 0,C 180,E1 24631.392,E2 24631.392} C_VEL
LIN {X 0,Y 537.558,Z 278.96,A -85,B 0,C 180,E1 24628.488,E2 24628.488} C_VEL
LIN {X 0,Y 537.556,Z 278.967,A -85,B 0,C 180,E1 24625.047,E2 24625.047} C_VEL
LIN {X 0,Y 537.639,Z 279.404,A -85,B 0,C 180,E1 24624.22,E2 24624.22} C_VEL
LIN {X 0,Y 538.229,Z 281.265,A -85,B 0,C 180,E1 24623.97,E2 24623.97} C_VEL
LIN {X 0,Y 540.4,Z 284.145,A -85,B 0,C 180,E1 24623.563,E2 24623.563} C_VEL
LIN {X 0,Y 542.227,Z 285.837,A -85,B 0,C 180,E1 24623.245,E2 24623.245} C_VEL
LIN {X 0,Y 544.873,Z 289.661,A -85,B 0,C 180,E1 24622.762,E2 24622.762} C_VEL
LIN {X 0,Y 547.234,Z 292.292,A -85,B 0,C 180,E1 24622.357,E2 24622.357} C_VEL
LIN {X 0,Y 557.68,Z 306.281,A -85,B 0,C 180,E1 24620.602,E2 24620.602} C_VEL
LIN {X 0,Y 570.343,Z 324.04,A -85,B 0,C 180,E1 24618.629,E2 24618.629} C_VEL
LIN {X 0,Y 584.408,Z 345.371,A -85,B 0,C 180,E1 24616.594,E2 24616.594} C_VEL
LIN {X 0,Y 591.743,Z 357.151,A -85,B 0,C 180,E1 24615.585,E2 24615.585} C_VEL
LIN {X 0,Y 585.13,Z 574.053,A -85,B 0,C 180,E1 24612.513,E2 24612.513} C_VEL
LIN {X 0,Y 582.048,Z 679.958,A -85,B 0,C 180,E1 24611.032,E2 24611.032} C_VEL
LIN {X 0,Y 581.092,Z 687.656,A -85,B 0,C 180,E1 24610.995,E2 24610.995} C_VEL
LIN {X 0,Y 575.771,Z 708.195,A -85,B 0,C 180,E1 24611.12,E2 24611.12} C_VEL
LIN {X 0,Y 574.959,Z 714.781,A -85,B 0,C 180,E1 24611.064,E2 24611.064} C_VEL
LIN {X 0,Y 573.081,Z 741.911,A -85,B 0,C 180,E1 24610.511,E2 24610.511} C_VEL
LIN {X 0,Y 571.1,Z 763.96,A -85,B 0,C 180,E1 24609.909,E2 24609.909} C_VEL
LIN {X 0,Y 568.45,Z 788.917,A -85,B 0,C 180,E1 24609.061,E2 24609.061} C_VEL
LIN {X 0,Y 565.37,Z 812.672,A -85,B 0,C 180,E1 24608.049,E2 24608.049} C_VEL
LIN {X 0,Y 562.481,Z 832.767,A -85,B 0,C 180,E1 24607.045,E2 24607.045} C_VEL
LIN {X 0,Y 558.976,Z 855.485,A -85,B 0,C 180,E1 24605.725,E2 24605.725} C_VEL
LIN {X 0,Y 555.299,Z 876.829,A -85,B 0,C 180,E1 24604.26,E2 24604.26} C_VEL
LIN {X 0,Y 552.183,Z 894.233,A -85,B 0,C 180,E1 24602.904,E2 24602.904} C_VEL
LIN {X 0,Y 548.587,Z 913.897,A -85,B 0,C 180,E1 24601.174,E2 24601.174} C_VEL
LIN {X 0,Y 544.89,Z 933.116,A -85,B 0,C 180,E1 24599.217,E2 24599.217} C_VEL
LIN {X 0,Y 541.99,Z 948.408,A -85,B 0,C 180,E1 24597.454,E2 24597.454} C_VEL
LIN {X 0,Y 538.909,Z 965.344,A -85,B 0,C 180,E1 24595.261,E2 24595.261} C_VEL
LIN {X 0,Y 536.098,Z 980.83,A -85,B 0,C 180,E1 24592.943,E2 24592.943} C_VEL
LIN {X 0,Y 534.036,Z 993.262,A -85,B 0,C 180,E1 24590.839,E2 24590.839} C_VEL
LIN {X 0,Y 532.046,Z 1006.55,A -85,B 0,C 180,E1 24588.291,E2 24588.291} C_VEL
LIN {X 0,Y 530.529,Z 1017.785,A -85,B 0,C 180,E1 24585.747,E2 24585.747} C_VEL
LIN {X 0,Y 529.562,Z 1026.438,A -85,B 0,C 180,E1 24583.493,E2 24583.493} C_VEL
LIN {X 0,Y 528.781,Z 1035.313,A -85,B 0,C 180,E1 24580.789,E2 24580.789} C_VEL
LIN {X 0,Y 528.285,Z 1042.231,A -85,B 0,C 180,E1 24578.153,E2 24578.153} C_VEL
LIN {X 0,Y 528.056,Z 1047.07,A -85,B 0,C 180,E1 24575.869,E2 24575.869} C_VEL
LIN {X 0,Y 527.961,Z 1050.812,A -85,B 0,C 180,E1 24573.583,E2 24573.583} C_VEL
LIN {X 0,Y 527.921,Z 1053.956,A -85,B 0,C 180,E1 24570.76,E2 24570.76} C_VEL
LIN {X 0,Y 527.907,Z 1055.256,A -85,B 0,C 180,E1 24568.155,E2 24568.155} C_VEL
LIN {X 0,Y 527.905,Z 1055.303,A -85,B 0,C 180,E1 24565.981,E2 24565.981} C_VEL
LIN {X 0,Y 527.912,Z 1054.297,A -85,B 0,C 180,E1 24563.693,E2 24563.693} C_VEL
LIN {X 0,Y 527.93,Z 1051.858,A -85,B 0,C 180,E1 24561.065,E2 24561.065} C_VEL
LIN {X 0,Y 528.042,Z 1047.577,A -85,B 0,C 180,E1 24558.31,E2 24558.31} C_VEL
LIN {X 0,Y 528.26,Z 1042.744,A -85,B 0,C 180,E1 24555.979,E2 24555.979} C_VEL
LIN {X 0,Y 528.647,Z 1036.711,A -85,B 0,C 180,E1 24553.631,E2 24553.631} C_VEL
LIN {X 0,Y 529.452,Z 1027.468,A -85,B 0,C 180,E1 24550.701,E2 24550.701} C_VEL
LIN {X 0,Y 530.453,Z 1018.417,A -85,B 0,C 180,E1 24548.318,E2 24548.318} C_VEL
LIN {X 0,Y 531.837,Z 1007.934,A -85,B 0,C 180,E1 24545.922,E2 24545.922} C_VEL
LIN {X 0,Y 533.86,Z 994.481,A -85,B 0,C 180,E1 24543.288,E2 24543.288} C_VEL
LIN {X 0,Y 535.824,Z 982.408,A -85,B 0,C 180,E1 24541.22,E2 24541.22} C_VEL
LIN {X 0,Y 538.297,Z 968.568,A -85,B 0,C 180,E1 24539.112,E2 24539.112} C_VEL
LIN {X 0,Y 541.648,Z 950.341,A -85,B 0,C 180,E1 24536.689,E2 24536.689} C_VEL
LIN {X 0,Y 544.603,Z 934.66,A -85,B 0,C 180,E1 24534.86,E2 24534.86} C_VEL
LIN {X 0,Y 548.225,Z 916.057,A -85,B 0,C 180,E1 24532.93,E2 24532.93} C_VEL
LIN {X 0,Y 552.122,Z 895.273,A -85,B 0,C 180,E1 24531.067,E2 24531.067} C_VEL
LIN {X 0,Y 555.375,Z 877.528,A -85,B 0,C 180,E1 24529.666,E2 24529.666} C_VEL
LIN {X 0,Y 559.019,Z 856.942,A -85,B 0,C 180,E1 24528.234,E2 24528.234} C_VEL
LIN {X 0,Y 562.787,Z 833.436,A -85,B 0,C 180,E1 24526.842,E2 24526.842} C_VEL
LIN {X 0,Y 565.686,Z 814.072,A -85,B 0,C 180,E1 24525.86,E2 24525.86} C_VEL
LIN {X 0,Y 568.63,Z 792.306,A -85,B 0,C 180,E1 24524.911,E2 24524.911} C_VEL
LIN {X 0,Y 571.632,Z 765.922,A -85,B 0,C 180,E1 24523.978,E2 24523.978} C_VEL
LIN {X 0,Y 573.702,Z 744.033,A -85,B 0,C 180,E1 24523.365,E2 24523.365} C_VEL
LIN {X 0,Y 575.577,Z 719.546,A -85,B 0,C 180,E1 24522.835,E2 24522.835} C_VEL
LIN {X 0,Y 577.135,Z 681.158,A -85,B 0,C 180,E1 24522.252,E2 24522.252} C_VEL
LIN {X 0,Y 584.766,Z 452.993,A -85,B 0,C 180,E1 24518.982,E2 24518.982} C_VEL
LIN {X 0,Y 587.916,Z 360.757,A -85,B 0,C 180,E1 24517.631,E2 24517.631} C_VEL
LIN {X 0,Y 577.628,Z 344.618,A -85,B 0,C 180,E1 24516.054,E2 24516.054} C_VEL
LIN {X 0,Y 565.753,Z 327.15,A -85,B 0,C 180,E1 24514.104,E2 24514.104} C_VEL
LIN {X 0,Y 554.348,Z 311.719,A -85,B 0,C 180,E1 24512.087,E2 24512.087} C_VEL
LIN {X 0,Y 546.888,Z 302.117,A -85,B 0,C 180,E1 24510.671,E2 24510.671} C_VEL
LIN {X 0,Y 543.024,Z 297.314,A -85,B 0,C 180,E1 24509.904,E2 24509.904} C_VEL
LIN {X 0,Y 539.841,Z 293.072,A -85,B 0,C 180,E1 24509.243,E2 24509.243} C_VEL
LIN {X 0,Y 535.946,Z 289.121,A -85,B 0,C 180,E1 24508.438,E2 24508.438} C_VEL
LIN {X 0,Y 534.375,Z 286.368,A -85,B 0,C 180,E1 24508.073,E2 24508.073} C_VEL
LIN {X 0,Y 531.216,Z 283.854,A -85,B 0,C 180,E1 24507.401,E2 24507.401} C_VEL
LIN {X 0,Y 529.719,Z 280.592,A -85,B 0,C 180,E1 24506.938,E2 24506.938} C_VEL
LIN {X 0,Y 529.643,Z 279.952,A -85,B 0,C 180,E1 24506.458,E2 24506.458} C_VEL
LIN {X 0,Y 529.619,Z 280.008,A -85,B 0,C 180,E1 24503.122,E2 24503.122} C_VEL
LIN {X 0,Y 529.668,Z 279.929,A -85,B 0,C 180,E1 24499.865,E2 24499.865} C_VEL
LIN {X 0,Y 529.629,Z 280.006,A -85,B 0,C 180,E1 24496.563,E2 24496.563} C_VEL
LIN {X 0,Y 529.612,Z 279.935,A -85,B 0,C 180,E1 24493.094,E2 24493.094} C_VEL
LIN {X 0,Y 529.678,Z 279.994,A -85,B 0,C 180,E1 24489.782,E2 24489.782} C_VEL
LIN {X 0,Y 529.614,Z 279.927,A -85,B 0,C 180,E1 24486.504,E2 24486.504} C_VEL
LIN {X 0,Y 529.626,Z 280.004,A -85,B 0,C 180,E1 24483.03,E2 24483.03} C_VEL
LIN {X 0,Y 529.682,Z 279.92,A -85,B 0,C 180,E1 24479.676,E2 24479.676} C_VEL
LIN {X 0,Y 529.625,Z 280.01,A -85,B 0,C 180,E1 24476.32,E2 24476.32} C_VEL
LIN {X 0,Y 529.617,Z 279.925,A -85,B 0,C 180,E1 24472.842,E2 24472.842} C_VEL
LIN {X 0,Y 529.676,Z 280,A -85,B 0,C 180,E1 24469.559,E2 24469.559} C_VEL
LIN {X 0,Y 529.611,Z 279.926,A -85,B 0,C 180,E1 24466.238,E2 24466.238} C_VEL
LIN {X 0,Y 529.632,Z 280.004,A -85,B 0,C 180,E1 24462.758,E2 24462.758} C_VEL
LIN {X 0,Y 529.669,Z 279.926,A -85,B 0,C 180,E1 24459.443,E2 24459.443} C_VEL
LIN {X 0,Y 529.621,Z 280.003,A -85,B 0,C 180,E1 24456.17,E2 24456.17} C_VEL
LIN {X 0,Y 529.646,Z 279.997,A -85,B 0,C 180,E1 24452.769,E2 24452.769} C_VEL
LIN {X 0,Y 529.691,Z 280.288,A -85,B 0,C 180,E1 24450.762,E2 24450.762} C_VEL
LIN {X 0,Y 531.031,Z 283.635,A -85,B 0,C 180,E1 24449.943,E2 24449.943} C_VEL
LIN {X 0,Y 532.532,Z 285.694,A -85,B 0,C 180,E1 24449.414,E2 24449.414} C_VEL
LIN {X 0,Y 535.734,Z 289.964,A -85,B 0,C 180,E1 24448.682,E2 24448.682} C_VEL
LIN {X 0,Y 543.447,Z 299.658,A -85,B 0,C 180,E1 24447.064,E2 24447.064} C_VEL
LIN {X 0,Y 549.81,Z 307.968,A -85,B 0,C 180,E1 24445.809,E2 24445.809} C_VEL
LIN {X 0,Y 559.118,Z 320.487,A -85,B 0,C 180,E1 24444.086,E2 24444.086} C_VEL
LIN {X 0,Y 567.78,Z 332.824,A -85,B 0,C 180,E1 24442.586,E2 24442.586} C_VEL
LIN {X 0,Y 578.622,Z 348.885,A -85,B 0,C 180,E1 24440.831,E2 24440.831} C_VEL
LIN {X 0,Y 588.073,Z 364.314,A -85,B 0,C 180,E1 24439.379,E2 24439.379} C_VEL
LIN {X 0,Y 580.094,Z 594.414,A -85,B 0,C 180,E1 24436.064,E2 24436.064} C_VEL
LIN {X 0,Y 575.841,Z 720.259,A -85,B 0,C 180,E1 24434.252,E2 24434.252} C_VEL
LIN {X 0,Y 573.969,Z 747.487,A -85,B 0,C 180,E1 24433.717,E2 24433.717} C_VEL
LIN {X 0,Y 571.798,Z 770.712,A -85,B 0,C 180,E1 24433.093,E2 24433.093} C_VEL
LIN {X 0,Y 569.488,Z 791.714,A -85,B 0,C 180,E1 24432.393,E2 24432.393} C_VEL
LIN {X 0,Y 566.243,Z 816.947,A -85,B 0,C 180,E1 24431.368,E2 24431.368} C_VEL
LIN {X 0,Y 562.971,Z 839.058,A -85,B 0,C 180,E1 24430.278,E2 24430.278} C_VEL
LIN {X 0,Y 559.854,Z 858.693,A -85,B 0,C 180,E1 24429.156,E2 24429.156} C_VEL
LIN {X 0,Y 555.795,Z 882.424,A -85,B 0,C 180,E1 24427.58,E2 24427.58} C_VEL
LIN {X 0,Y 552.326,Z 901.53,A -85,B 0,C 180,E1 24426.104,E2 24426.104} C_VEL
LIN {X 0,Y 548.931,Z 919.857,A -85,B 0,C 180,E1 24424.506,E2 24424.506} C_VEL
LIN {X 0,Y 544.843,Z 941.473,A -85,B 0,C 180,E1 24422.341,E2 24422.341} C_VEL
LIN {X 0,Y 541.819,Z 957.59,A -85,B 0,C 180,E1 24420.497,E2 24420.497} C_VEL
LIN {X 0,Y 538.84,Z 974.206,A -85,B 0,C 180,E1 24418.362,E2 24418.362} C_VEL
LIN {X 0,Y 536.015,Z 990.156,A -85,B 0,C 180,E1 24416,E2 24416} C_VEL
LIN {X 0,Y 533.941,Z 1002.916,A -85,B 0,C 180,E1 24413.859,E2 24413.859} C_VEL
LIN {X 0,Y 531.954,Z 1016.497,A -85,B 0,C 180,E1 24411.271,E2 24411.271} C_VEL
LIN {X 0,Y 530.511,Z 1027.517,A -85,B 0,C 180,E1 24408.802,E2 24408.802} C_VEL
LIN {X 0,Y 529.562,Z 1036.216,A -85,B 0,C 180,E1 24406.565,E2 24406.565} C_VEL
LIN {X 0,Y 528.791,Z 1045.119,A -85,B 0,C 180,E1 24403.895,E2 24403.895} C_VEL
LIN {X 0,Y 528.29,Z 1052.131,A -85,B 0,C 180,E1 24401.242,E2 24401.242} C_VEL
LIN {X 0,Y 528.057,Z 1057.035,A -85,B 0,C 180,E1 24398.932,E2 24398.932} C_VEL
LIN {X 0,Y 527.964,Z 1060.645,A -85,B 0,C 180,E1 24396.743,E2 24396.743} C_VEL
LIN {X 0,Y 527.915,Z 1063.808,A -85,B 0,C 180,E1 24394.019,E2 24394.019} C_VEL
LIN {X 0,Y 527.907,Z 1065.235,A -85,B 0,C 180,E1 24391.302,E2 24391.302} C_VEL
LIN {X 0,Y 527.905,Z 1065.325,A -85,B 0,C 180,E1 24389.132,E2 24389.132} C_VEL
LIN {X 0,Y 527.912,Z 1064.367,A -85,B 0,C 180,E1 24386.851,E2 24386.851} C_VEL
LIN {X 0,Y 527.922,Z 1062.218,A -85,B 0,C 180,E1 24384.457,E2 24384.457} C_VEL
LIN {X 0,Y 528.035,Z 1058.067,A -85,B 0,C 180,E1 24381.616,E2 24381.616} C_VEL
LIN {X 0,Y 528.243,Z 1053.148,A -85,B 0,C 180,E1 24379.199,E2 24379.199} C_VEL
LIN {X 0,Y 528.588,Z 1047.472,A -85,B 0,C 180,E1 24376.955,E2 24376.955} C_VEL
LIN {X 0,Y 529.227,Z 1039.786,A -85,B 0,C 180,E1 24374.438,E2 24374.438} C_VEL
LIN {X 0,Y 530.246,Z 1029.832,A -85,B 0,C 180,E1 24371.758,E2 24371.758} C_VEL
LIN {X 0,Y 531.452,Z 1020.133,A -85,B 0,C 180,E1 24369.516,E2 24369.516} C_VEL
LIN {X 0,Y 533.095,Z 1008.495,A -85,B 0,C 180,E1 24367.154,E2 24367.154} C_VEL
LIN {X 0,Y 535.435,Z 993.69,A -85,B 0,C 180,E1 24364.564,E2 24364.564} C_VEL
LIN {X 0,Y 537.73,Z 980.205,A -85,B 0,C 180,E1 24362.495,E2 24362.495} C_VEL
LIN {X 0,Y 540.688,Z 964.037,A -85,B 0,C 180,E1 24360.29,E2 24360.29} C_VEL
LIN {X 0,Y 544.055,Z 945.627,A -85,B 0,C 180,E1 24358.113,E2 24358.113} C_VEL
LIN {X 0,Y 546.992,Z 929.91,A -85,B 0,C 180,E1 24356.467,E2 24356.467} C_VEL
LIN {X 0,Y 550.631,Z 910.538,A -85,B 0,C 180,E1 24354.665,E2 24354.665} C_VEL
LIN {X 0,Y 554.417,Z 889.274,A -85,B 0,C 180,E1 24352.961,E2 24352.961} C_VEL
LIN {X 0,Y 557.467,Z 871.477,A -85,B 0,C 180,E1 24351.706,E2 24351.706} C_VEL
LIN {X 0,Y 560.736,Z 851.435,A -85,B 0,C 180,E1 24350.462,E2 24350.462} C_VEL
LIN {X 0,Y 564.412,Z 826.633,A -85,B 0,C 180,E1 24349.153,E2 24349.153} C_VEL
LIN {X 0,Y 567.074,Z 806.632,A -85,B 0,C 180,E1 24348.263,E2 24348.263} C_VEL
LIN {X 0,Y 569.385,Z 787.187,A -85,B 0,C 180,E1 24347.524,E2 24347.524} C_VEL
LIN {X 0,Y 571.817,Z 763.878,A -85,B 0,C 180,E1 24346.789,E2 24346.789} C_VEL
LIN {X 0,Y 573.892,Z 738.144,A -85,B 0,C 180,E1 24346.171,E2 24346.171} C_VEL
LIN {X 0,Y 575.151,Z 716.295,A -85,B 0,C 180,E1 24345.778,E2 24345.778} C_VEL
LIN {X 0,Y 582.404,Z 483.832,A -85,B 0,C 180,E1 24342.483,E2 24342.483} C_VEL
LIN {X 0,Y 586.14,Z 363.602,A -85,B 0,C 180,E1 24340.749,E2 24340.749} C_VEL
LIN {X 0,Y 571.597,Z 340.612,A -85,B 0,C 180,E1 24338.662,E2 24338.662} C_VEL
LIN {X 0,Y 558.494,Z 321.138,A -85,B 0,C 180,E1 24336.629,E2 24336.629} C_VEL
LIN {X 0,Y 549.31,Z 308.466,A -85,B 0,C 180,E1 24335.114,E2 24335.114} C_VEL
LIN {X 0,Y 541.845,Z 298.324,A -85,B 0,C 180,E1 24333.805,E2 24333.805} C_VEL
LIN {X 0,Y 534.715,Z 289.101,A -85,B 0,C 180,E1 24332.49,E2 24332.49} C_VEL
LIN {X 0,Y 532.107,Z 285.354,A -85,B 0,C 180,E1 24331.936,E2 24331.936} C_VEL
LIN {X 0,Y 529.9,Z 281.122,A -85,B 0,C 180,E1 24331.007,E2 24331.007} C_VEL
LIN {X 0,Y 529.708,Z 280.143,A -85,B 0,C 180,E1 24330.767,E2 24330.767} C_VEL
LIN {X 0,Y 529.619,Z 279.948,A -85,B 0,C 180,E1 24327.552,E2 24327.552} C_VEL
LIN {X 0,Y 529.625,Z 279.987,A -85,B 0,C 180,E1 24324.066,E2 24324.066} C_VEL
LIN {X 0,Y 529.672,Z 279.984,A -85,B 0,C 180,E1 24320.864,E2 24320.864} C_VEL
LIN {X 0,Y 529.619,Z 279.998,A -85,B 0,C 180,E1 24317.56,E2 24317.56} C_VEL
LIN {X 0,Y 529.65,Z 280.004,A -85,B 0,C 180,E1 24314.207,E2 24314.207} C_VEL
LIN {X 0,Y 529.642,Z 280.002,A -85,B 0,C 180,E1 24310.984,E2 24310.984} C_VEL
LIN {X 0,Y 529.616,Z 279.991,A -85,B 0,C 180,E1 24307.594,E2 24307.594} C_VEL
LIN {X 0,Y 529.673,Z 279.977,A -85,B 0,C 180,E1 24304.331,E2 24304.331} C_VEL
LIN {X 0,Y 529.625,Z 279.998,A -85,B 0,C 180,E1 24301.082,E2 24301.082} C_VEL
LIN {X 0,Y 529.625,Z 280.008,A -85,B 0,C 180,E1 24297.62,E2 24297.62} C_VEL
LIN {X 0,Y 529.683,Z 279.989,A -85,B 0,C 180,E1 24294.258,E2 24294.258} C_VEL
LIN {X 0,Y 529.619,Z 279.982,A -85,B 0,C 180,E1 24290.985,E2 24290.985} C_VEL
LIN {X 0,Y 529.629,Z 279.983,A -85,B 0,C 180,E1 24287.571,E2 24287.571} C_VEL
LIN {X 0,Y 529.663,Z 279.995,A -85,B 0,C 180,E1 24284.338,E2 24284.338} C_VEL
LIN {X 0,Y 529.619,Z 280.009,A -85,B 0,C 180,E1 24281.051,E2 24281.051} C_VEL
LIN {X 0,Y 529.659,Z 279.997,A -85,B 0,C 180,E1 24277.7,E2 24277.7} C_VEL
LIN {X 0,Y 529.623,Z 279.921,A -85,B 0,C 180,E1 24274.478,E2 24274.478} C_VEL
LIN {X 0,Y 529.618,Z 279.971,A -85,B 0,C 180,E1 24271.098,E2 24271.098} C_VEL
LIN {X 0,Y 529.652,Z 279.93,A -85,B 0,C 180,E1 24268.09,E2 24268.09} C_VEL
LIN {X 0,Y 529.688,Z 280.176,A -85,B 0,C 180,E1 24265.544,E2 24265.544} C_VEL
LIN {X 0,Y 529.818,Z 280.908,A -85,B 0,C 180,E1 24265.369,E2 24265.369} C_VEL
LIN {X 0,Y 531.586,Z 284.299,A -85,B 0,C 180,E1 24264.959,E2 24264.959} C_VEL
LIN {X 0,Y 534.442,Z 286.814,A -85,B 0,C 180,E1 24264.435,E2 24264.435} C_VEL
LIN {X 0,Y 537.065,Z 290.692,A -85,B 0,C 180,E1 24263.929,E2 24263.929} C_VEL
LIN {X 0,Y 539.124,Z 292.759,A -85,B 0,C 180,E1 24263.562,E2 24263.562} C_VEL
LIN {X 0,Y 542.283,Z 296.947,A -85,B 0,C 180,E1 24262.985,E2 24262.985} C_VEL
LIN {X 0,Y 546.966,Z 302.897,A -85,B 0,C 180,E1 24262.163,E2 24262.163} C_VEL
LIN {X 0,Y 557.952,Z 317.93,A -85,B 0,C 180,E1 24260.325,E2 24260.325} C_VEL
LIN {X 0,Y 569.868,Z 335.265,A -85,B 0,C 180,E1 24258.469,E2 24258.469} C_VEL
LIN {X 0,Y 581.411,Z 353.002,A -85,B 0,C 180,E1 24256.789,E2 24256.789} C_VEL
LIN {X 0,Y 586.239,Z 360.865,A -85,B 0,C 180,E1 24256.112,E2 24256.112} C_VEL
LIN {X 0,Y 579.378,Z 576.115,A -85,B 0,C 180,E1 24253.041,E2 24253.041} C_VEL
LIN {X 0,Y 575.085,Z 711.979,A -85,B 0,C 180,E1 24251.109,E2 24251.109} C_VEL
LIN {X 0,Y 574.959,Z 714.781,A -85,B 0,C 180,E1 24251.064,E2 24251.064} C_VEL
LIN {X 0,Y 573.842,Z 722.435,A -85,B 0,C 180,E1 24250.998,E2 24250.998} C_VEL
LIN {X 0,Y 568.241,Z 740.602,A -85,B 0,C 180,E1 24251.006,E2 24251.006} C_VEL
LIN {X 0,Y 566.712,Z 748.132,A -85,B 0,C 180,E1 24250.901,E2 24250.901} C_VEL
LIN {X 0,Y 566.607,Z 749.206,A -85,B 0,C 180,E1 24250.875,E2 24250.875} C_VEL
LIN {X 0,Y 563.996,Z 775.312,A -85,B 0,C 180,E1 24250.09,E2 24250.09} C_VEL
LIN {X 0,Y 561.551,Z 795.45,A -85,B 0,C 180,E1 24249.337,E2 24249.337} C_VEL
LIN {X 0,Y 558.791,Z 815.64,A -85,B 0,C 180,E1 24248.448,E2 24248.448} C_VEL
LIN {X 0,Y 555.386,Z 838.406,A -85,B 0,C 180,E1 24247.273,E2 24247.273} C_VEL
LIN {X 0,Y 551.539,Z 861.218,A -85,B 0,C 180,E1 24245.867,E2 24245.867} C_VEL
LIN {X 0,Y 548.344,Z 879.018,A -85,B 0,C 180,E1 24244.611,E2 24244.611} C_VEL
LIN {X 0,Y 544.802,Z 898.029,A -85,B 0,C 180,E1 24243.093,E2 24243.093} C_VEL
LIN {X 0,Y 540.615,Z 919.412,A -85,B 0,C 180,E1 24241.121,E2 24241.121} C_VEL
LIN {X 0,Y 537.399,Z 935.568,A -85,B 0,C 180,E1 24239.419,E2 24239.419} C_VEL
LIN {X 0,Y 534.109,Z 952.415,A -85,B 0,C 180,E1 24237.421,E2 24237.421} C_VEL
LIN {X 0,Y 530.774,Z 969.563,A -85,B 0,C 180,E1 24235.078,E2 24235.078} C_VEL
LIN {X 0,Y 528.332,Z 982.581,A -85,B 0,C 180,E1 24233.064,E2 24233.064} C_VEL
LIN {X 0,Y 526.021,Z 996.101,A -85,B 0,C 180,E1 24230.705,E2 24230.705} C_VEL
LIN {X 0,Y 523.912,Z 1009.372,A -85,B 0,C 180,E1 24228.01,E2 24228.01} C_VEL
LIN {X 0,Y 522.579,Z 1019.002,A -85,B 0,C 180,E1 24225.755,E2 24225.755} C_VEL
LIN {X 0,Y 521.518,Z 1028.111,A -85,B 0,C 180,E1 24223.301,E2 24223.301} C_VEL
LIN {X 0,Y 520.69,Z 1037.016,A -85,B 0,C 180,E1 24220.399,E2 24220.399} C_VEL
LIN {X 0,Y 520.284,Z 1042.861,A -85,B 0,C 180,E1 24218.065,E2 24218.065} C_VEL
LIN {X 0,Y 520.051,Z 1047.57,A -85,B 0,C 180,E1 24215.738,E2 24215.738} C_VEL
LIN {X 0,Y 519.938,Z 1051.814,A -85,B 0,C 180,E1 24212.976,E2 24212.976} C_VEL
LIN {X 0,Y 519.919,Z 1054.256,A -85,B 0,C 180,E1 24210.331,E2 24210.331} C_VEL
LIN {X 0,Y 519.908,Z 1055.288,A -85,B 0,C 180,E1 24208.016,E2 24208.016} C_VEL
LIN {X 0,Y 519.906,Z 1055.248,A -85,B 0,C 180,E1 24205.698,E2 24205.698} C_VEL
LIN {X 0,Y 519.923,Z 1053.925,A -85,B 0,C 180,E1 24203.041,E2 24203.041} C_VEL
LIN {X 0,Y 519.963,Z 1050.861,A -85,B 0,C 180,E1 24200.257,E2 24200.257} C_VEL
LIN {X 0,Y 520.072,Z 1047.075,A -85,B 0,C 180,E1 24197.903,E2 24197.903} C_VEL
LIN {X 0,Y 520.327,Z 1042.158,A -85,B 0,C 180,E1 24195.533,E2 24195.533} C_VEL
LIN {X 0,Y 520.901,Z 1034.735,A -85,B 0,C 180,E1 24192.691,E2 24192.691} C_VEL
LIN {X 0,Y 521.698,Z 1026.552,A -85,B 0,C 180,E1 24190.17,E2 24190.17} C_VEL
LIN {X 0,Y 522.736,Z 1017.831,A -85,B 0,C 180,E1 24187.863,E2 24187.863} C_VEL
LIN {X 0,Y 524.437,Z 1006.042,A -85,B 0,C 180,E1 24185.168,E2 24185.168} C_VEL
LIN {X 0,Y 526.419,Z 993.538,A -85,B 0,C 180,E1 24182.74,E2 24182.74} C_VEL
LIN {X 0,Y 528.544,Z 981.463,A -85,B 0,C 180,E1 24180.661,E2 24180.661} C_VEL
LIN {X 0,Y 531.605,Z 965.415,A -85,B 0,C 180,E1 24178.221,E2 24178.221} C_VEL
LIN {X 0,Y 534.845,Z 948.613,A -85,B 0,C 180,E1 24176.015,E2 24176.015} C_VEL
LIN {X 0,Y 538.155,Z 932.232,A -85,B 0,C 180,E1 24174.105,E2 24174.105} C_VEL
LIN {X 0,Y 542.329,Z 911.487,A -85,B 0,C 180,E1 24171.991,E2 24171.991} C_VEL
LIN {X 0,Y 545.855,Z 893.548,A -85,B 0,C 180,E1 24170.397,E2 24170.397} C_VEL
LIN {X 0,Y 549.432,Z 874.893,A -85,B 0,C 180,E1 24168.931,E2 24168.931} C_VEL
LIN {X 0,Y 553.79,Z 850.706,A -85,B 0,C 180,E1 24167.295,E2 24167.295} C_VEL
LIN {X 0,Y 557.079,Z 830.858,A -85,B 0,C 180,E1 24166.146,E2 24166.146} C_VEL
LIN {X 0,Y 560.472,Z 808.879,A -85,B 0,C 180,E1 24165.052,E2 24165.052} C_VEL
LIN {X 0,Y 563.821,Z 783.73,A -85,B 0,C 180,E1 24164.018,E2 24164.018} C_VEL
LIN {X 0,Y 566.251,Z 762.317,A -85,B 0,C 180,E1 24163.299,E2 24163.299} C_VEL
LIN {X 0,Y 568.538,Z 738.407,A -85,B 0,C 180,E1 24162.654,E2 24162.654} C_VEL
LIN {X 0,Y 570.357,Z 711.982,A -85,B 0,C 180,E1 24162.136,E2 24162.136} C_VEL
LIN {X 0,Y 576.901,Z 526.809,A -85,B 0,C 180,E1 24159.454,E2 24159.454} C_VEL
LIN {X 0,Y 582.646,Z 364.494,A -85,B 0,C 180,E1 24157.07,E2 24157.07} C_VEL
LIN {X 0,Y 573.431,Z 350.024,A -85,B 0,C 180,E1 24155.619,E2 24155.619} C_VEL
LIN {X 0,Y 562.206,Z 333.352,A -85,B 0,C 180,E1 24153.734,E2 24153.734} C_VEL
LIN {X 0,Y 551.048,Z 318.129,A -85,B 0,C 180,E1 24151.72,E2 24151.72} C_VEL
LIN {X 0,Y 543.791,Z 308.702,A -85,B 0,C 180,E1 24150.314,E2 24150.314} C_VEL
LIN {X 0,Y 540.2,Z 304.207,A -85,B 0,C 180,E1 24149.587,E2 24149.587} C_VEL
LIN {X 0,Y 536.471,Z 299.444,A -85,B 0,C 180,E1 24148.803,E2 24148.803} C_VEL
LIN {X 0,Y 533.208,Z 295.995,A -85,B 0,C 180,E1 24148.109,E2 24148.109} C_VEL
LIN {X 0,Y 531.628,Z 293.511,A -85,B 0,C 180,E1 24147.743,E2 24147.743} C_VEL
LIN {X 0,Y 528.431,Z 290.575,A -85,B 0,C 180,E1 24147.039,E2 24147.039} C_VEL
LIN {X 0,Y 526.521,Z 287.368,A -85,B 0,C 180,E1 24146.566,E2 24146.566} C_VEL
LIN {X 0,Y 523.303,Z 284.802,A -85,B 0,C 180,E1 24145.827,E2 24145.827} C_VEL
LIN {X 0,Y 521.84,Z 281.82,A -85,B 0,C 180,E1 24145.381,E2 24145.381} C_VEL
LIN {X 0,Y 521.679,Z 280.983,A -85,B 0,C 180,E1 24144.94,E2 24144.94} C_VEL
LIN {X 0,Y 521.702,Z 280.944,A -85,B 0,C 180,E1 24141.592,E2 24141.592} C_VEL
LIN {X 0,Y 521.707,Z 280.946,A -85,B 0,C 180,E1 24138.32,E2 24138.32} C_VEL
LIN {X 0,Y 521.672,Z 280.935,A -85,B 0,C 180,E1 24134.981,E2 24134.981} C_VEL
LIN {X 0,Y 521.726,Z 280.951,A -85,B 0,C 180,E1 24131.67,E2 24131.67} C_VEL
LIN {X 0,Y 521.679,Z 280.934,A -85,B 0,C 180,E1 24128.487,E2 24128.487} C_VEL
LIN {X 0,Y 521.678,Z 280.951,A -85,B 0,C 180,E1 24124.948,E2 24124.948} C_VEL
LIN {X 0,Y 521.736,Z 280.932,A -85,B 0,C 180,E1 24121.647,E2 24121.647} C_VEL
LIN {X 0,Y 521.68,Z 280.94,A -85,B 0,C 180,E1 24118.353,E2 24118.353} C_VEL
LIN {X 0,Y 521.686,Z 280.949,A -85,B 0,C 180,E1 24114.942,E2 24114.942} C_VEL
LIN {X 0,Y 521.72,Z 280.92,A -85,B 0,C 180,E1 24111.736,E2 24111.736} C_VEL
LIN {X 0,Y 521.677,Z 280.965,A -85,B 0,C 180,E1 24108.502,E2 24108.502} C_VEL
LIN {X 0,Y 521.712,Z 280.918,A -85,B 0,C 180,E1 24105.119,E2 24105.119} C_VEL
LIN {X 0,Y 521.694,Z 280.964,A -85,B 0,C 180,E1 24101.911,E2 24101.911} C_VEL
LIN {X 0,Y 521.678,Z 280.932,A -85,B 0,C 180,E1 24098.525,E2 24098.525} C_VEL
LIN {X 0,Y 521.738,Z 280.97,A -85,B 0,C 180,E1 24095.285,E2 24095.285} C_VEL
LIN {X 0,Y 521.714,Z 281.204,A -85,B 0,C 180,E1 24092.306,E2 24092.306} C_VEL
LIN {X 0,Y 523.246,Z 284.741,A -85,B 0,C 180,E1 24091.338,E2 24091.338} C_VEL
LIN {X 0,Y 525.233,Z 287.277,A -85,B 0,C 180,E1 24090.802,E2 24090.802} C_VEL
LIN {X 0,Y 528.484,Z 291.251,A -85,B 0,C 180,E1 24090.034,E2 24090.034} C_VEL
LIN {X 0,Y 530.098,Z 293.11,A -85,B 0,C 180,E1 24089.666,E2 24089.666} C_VEL
LIN {X 0,Y 533.687,Z 297.557,A -85,B 0,C 180,E1 24088.862,E2 24088.862} C_VEL
LIN {X 0,Y 543.646,Z 310.521,A -85,B 0,C 180,E1 24086.764,E2 24086.764} C_VEL
LIN {X 0,Y 547.527,Z 315.747,A -85,B 0,C 180,E1 24085.994,E2 24085.994} C_VEL
LIN {X 0,Y 554.926,Z 325.686,A -85,B 0,C 180,E1 24084.599,E2 24084.599} C_VEL
LIN {X 0,Y 563.969,Z 338.649,A -85,B 0,C 180,E1 24082.992,E2 24082.992} C_VEL
LIN {X 0,Y 574.931,Z 355.062,A -85,B 0,C 180,E1 24081.18,E2 24081.18} C_VEL
LIN {X 0,Y 582.852,Z 368.125,A -85,B 0,C 180,E1 24079.932,E2 24079.932} C_VEL
LIN {X 0,Y 574.501,Z 598.971,A -85,B 0,C 180,E1 24076.584,E2 24076.584} C_VEL
LIN {X 0,Y 570.217,Z 720.205,A -85,B 0,C 180,E1 24074.825,E2 24074.825} C_VEL
LIN {X 0,Y 568.271,Z 747.522,A -85,B 0,C 180,E1 24074.285,E2 24074.285} C_VEL
LIN {X 0,Y 566.037,Z 770.582,A -85,B 0,C 180,E1 24073.663,E2 24073.663} C_VEL
LIN {X 0,Y 563.67,Z 791.308,A -85,B 0,C 180,E1 24072.97,E2 24072.97} C_VEL
LIN {X 0,Y 560.473,Z 815.524,A -85,B 0,C 180,E1 24071.99,E2 24071.99} C_VEL
LIN {X 0,Y 556.97,Z 838.242,A -85,B 0,C 180,E1 24070.871,E2 24070.871} C_VEL
LIN {X 0,Y 553.695,Z 858.032,A -85,B 0,C 180,E1 24069.737,E2 24069.737} C_VEL
LIN {X 0,Y 549.602,Z 881.052,A -85,B 0,C 180,E1 24068.211,E2 24068.211} C_VEL
LIN {X 0,Y 545.705,Z 901.461,A -85,B 0,C 180,E1 24066.626,E2 24066.626} C_VEL
LIN {X 0,Y 542.126,Z 919.887,A -85,B 0,C 180,E1 24065.002,E2 24065.002} C_VEL
LIN {X 0,Y 537.886,Z 941.268,A -85,B 0,C 180,E1 24062.835,E2 24062.835} C_VEL
LIN {X 0,Y 534.749,Z 957.062,A -85,B 0,C 180,E1 24061.007,E2 24061.007} C_VEL
LIN {X 0,Y 531.651,Z 973.27,A -85,B 0,C 180,E1 24058.904,E2 24058.904} C_VEL
LIN {X 0,Y 528.674,Z 989.367,A -85,B 0,C 180,E1 24056.51,E2 24056.51} C_VEL
LIN {X 0,Y 526.431,Z 1002.193,A -85,B 0,C 180,E1 24054.341,E2 24054.341} C_VEL
LIN {X 0,Y 524.479,Z 1014.739,A -85,B 0,C 180,E1 24051.942,E2 24051.942} C_VEL
LIN {X 0,Y 522.758,Z 1026.973,A -85,B 0,C 180,E1 24049.207,E2 24049.207} C_VEL
LIN {X 0,Y 521.722,Z 1035.726,A -85,B 0,C 180,E1 24046.936,E2 24046.936} C_VEL
LIN {X 0,Y 520.924,Z 1043.972,A -85,B 0,C 180,E1 24044.45,E2 24044.45} C_VEL
LIN {X 0,Y 520.34,Z 1051.837,A -85,B 0,C 180,E1 24041.528,E2 24041.528} C_VEL
LIN {X 0,Y 520.085,Z 1056.824,A -85,B 0,C 180,E1 24039.182,E2 24039.182} C_VEL
LIN {X 0,Y 519.971,Z 1060.486,A -85,B 0,C 180,E1 24036.958,E2 24036.958} C_VEL
LIN {X 0,Y 519.906,Z 1063.355,A -85,B 0,C 180,E1 24034.523,E2 24034.523} C_VEL
LIN {X 0,Y 519.897,Z 1065.167,A -85,B 0,C 180,E1 24031.653,E2 24031.653} C_VEL
LIN {X 0,Y 519.901,Z 1065.348,A -85,B 0,C 180,E1 24029.229,E2 24029.229} C_VEL
LIN {X 0,Y 519.913,Z 1064.503,A -85,B 0,C 180,E1 24027.024,E2 24027.024} C_VEL
LIN {X 0,Y 519.923,Z 1062.672,A -85,B 0,C 180,E1 24024.814,E2 24024.814} C_VEL
LIN {X 0,Y 520.004,Z 1059.526,A -85,B 0,C 180,E1 24022.376,E2 24022.376} C_VEL
LIN {X 0,Y 520.214,Z 1054.142,A -85,B 0,C 180,E1 24019.479,E2 24019.479} C_VEL
LIN {X 0,Y 520.564,Z 1048.418,A -85,B 0,C 180,E1 24017.126,E2 24017.126} C_VEL
LIN {X 0,Y 521.128,Z 1041.674,A -85,B 0,C 180,E1 24014.821,E2 24014.821} C_VEL
LIN {X 0,Y 522.11,Z 1032.41,A -85,B 0,C 180,E1 24012.14,E2 24012.14} C_VEL
LIN {X 0,Y 523.55,Z 1021.088,A -85,B 0,C 180,E1 24009.427,E2 24009.427} C_VEL
LIN {X 0,Y 525.068,Z 1010.72,A -85,B 0,C 180,E1 24007.259,E2 24007.259} C_VEL
LIN {X 0,Y 527.355,Z 997.09,A -85,B 0,C 180,E1 24004.745,E2 24004.745} C_VEL
LIN {X 0,Y 530.005,Z 981.955,A -85,B 0,C 180,E1 24002.349,E2 24002.349} C_VEL
LIN {X 0,Y 532.699,Z 967.729,A -85,B 0,C 180,E1 24000.351,E2 24000.351} C_VEL
LIN {X 0,Y 536.172,Z 950.025,A -85,B 0,C 180,E1 23998.146,E2 23998.146} C_VEL
LIN {X 0,Y 539.699,Z 931.658,A -85,B 0,C 180,E1 23996.17,E2 23996.17} C_VEL
LIN {X 0,Y 543.125,Z 914.024,A -85,B 0,C 180,E1 23994.491,E2 23994.491} C_VEL
LIN {X 0,Y 547.413,Z 891.379,A -85,B 0,C 180,E1 23992.614,E2 23992.614} C_VEL
LIN {X 0,Y 550.869,Z 872.025,A -85,B 0,C 180,E1 23991.229,E2 23991.229} C_VEL
LIN {X 0,Y 554.105,Z 852.949,A -85,B 0,C 180,E1 23990.029,E2 23990.029} C_VEL
LIN {X 0,Y 557.867,Z 828.978,A -85,B 0,C 180,E1 23988.732,E2 23988.732} C_VEL
LIN {X 0,Y 560.919,Z 806.852,A -85,B 0,C 180,E1 23987.734,E2 23987.734} C_VEL
LIN {X 0,Y 563.292,Z 787.662,A -85,B 0,C 180,E1 23986.999,E2 23986.999} C_VEL
LIN {X 0,Y 565.653,Z 765.853,A -85,B 0,C 180,E1 23986.301,E2 23986.301} C_VEL
LIN {X 0,Y 567.917,Z 739.672,A -85,B 0,C 180,E1 23985.652,E2 23985.652} C_VEL
LIN {X 0,Y 569.288,Z 717.057,A -85,B 0,C 180,E1 23985.238,E2 23985.238} C_VEL
LIN {X 0,Y 576.745,Z 488.182,A -85,B 0,C 180,E1 23981.968,E2 23981.968} C_VEL
LIN {X 0,Y 580.717,Z 367.264,A -85,B 0,C 180,E1 23980.217,E2 23980.217} C_VEL
LIN {X 0,Y 566.216,Z 344.38,A -85,B 0,C 180,E1 23978.079,E2 23978.079} C_VEL
LIN {X 0,Y 552.819,Z 324.452,A -85,B 0,C 180,E1 23975.939,E2 23975.939} C_VEL
LIN {X 0,Y 542.385,Z 310.077,A -85,B 0,C 180,E1 23974.149,E2 23974.149} C_VEL
LIN {X 0,Y 535.971,Z 301.381,A -85,B 0,C 180,E1 23972.976,E2 23972.976} C_VEL
LIN {X 0,Y 531.042,Z 295.122,A -85,B 0,C 180,E1 23972.04,E2 23972.04} C_VEL
LIN {X 0,Y 527.68,Z 290.723,A -85,B 0,C 180,E1 23971.374,E2 23971.374} C_VEL
LIN {X 0,Y 524.515,Z 286.441,A -85,B 0,C 180,E1 23970.723,E2 23970.723} C_VEL
LIN {X 0,Y 522.275,Z 283.133,A -85,B 0,C 180,E1 23969.979,E2 23969.979} C_VEL
LIN {X 0,Y 521.715,Z 281.158,A -85,B 0,C 180,E1 23969.509,E2 23969.509} C_VEL
LIN {X 0,Y 521.719,Z 280.961,A -85,B 0,C 180,E1 23966.523,E2 23966.523} C_VEL
LIN {X 0,Y 521.698,Z 280.977,A -85,B 0,C 180,E1 23963.255,E2 23963.255} C_VEL
LIN {X 0,Y 521.681,Z 280.977,A -85,B 0,C 180,E1 23959.831,E2 23959.831} C_VEL
LIN {X 0,Y 521.732,Z 280.968,A -85,B 0,C 180,E1 23956.478,E2 23956.478} C_VEL
LIN {X 0,Y 521.684,Z 280.979,A -85,B 0,C 180,E1 23953.297,E2 23953.297} C_VEL
LIN {X 0,Y 521.686,Z 280.992,A -85,B 0,C 180,E1 23949.822,E2 23949.822} C_VEL
LIN {X 0,Y 521.75,Z 280.988,A -85,B 0,C 180,E1 23946.492,E2 23946.492} C_VEL
LIN {X 0,Y 521.687,Z 280.982,A -85,B 0,C 180,E1 23943.07,E2 23943.07} C_VEL
LIN {X 0,Y 521.679,Z 280.972,A -85,B 0,C 180,E1 23939.561,E2 23939.561} C_VEL
LIN {X 0,Y 521.734,Z 280.969,A -85,B 0,C 180,E1 23936.264,E2 23936.264} C_VEL
LIN {X 0,Y 521.685,Z 280.996,A -85,B 0,C 180,E1 23932.954,E2 23932.954} C_VEL
LIN {X 0,Y 521.683,Z 280.999,A -85,B 0,C 180,E1 23929.397,E2 23929.397} C_VEL
LIN {X 0,Y 521.741,Z 280.973,A -85,B 0,C 180,E1 23926.026,E2 23926.026} C_VEL
LIN {X 0,Y 521.686,Z 280.971,A -85,B 0,C 180,E1 23922.718,E2 23922.718} C_VEL
LIN {X 0,Y 521.68,Z 280.972,A -85,B 0,C 180,E1 23919.232,E2 23919.232} C_VEL
LIN {X 0,Y 521.736,Z 280.953,A -85,B 0,C 180,E1 23916.028,E2 23916.028} C_VEL
LIN {X 0,Y 521.671,Z 280.905,A -85,B 0,C 180,E1 23912.736,E2 23912.736} C_VEL
LIN {X 0,Y 521.696,Z 280.965,A -85,B 0,C 180,E1 23909.348,E2 23909.348} C_VEL
LIN {X 0,Y 521.696,Z 281.107,A -85,B 0,C 180,E1 23906.927,E2 23906.927} C_VEL
LIN {X 0,Y 522.023,Z 282.458,A -85,B 0,C 180,E1 23906.652,E2 23906.652} C_VEL
LIN {X 0,Y 523.912,Z 285.513,A -85,B 0,C 180,E1 23906.23,E2 23906.23} C_VEL
LIN {X 0,Y 526.557,Z 287.71,A -85,B 0,C 180,E1 23905.718,E2 23905.718} C_VEL
LIN {X 0,Y 528.951,Z 291.463,A -85,B 0,C 180,E1 23905.221,E2 23905.221} C_VEL
LIN {X 0,Y 531.511,Z 293.951,A -85,B 0,C 180,E1 23904.739,E2 23904.739} C_VEL
LIN {X 0,Y 534.643,Z 298.098,A -85,B 0,C 180,E1 23904.137,E2 23904.137} C_VEL
LIN {X 0,Y 536.393,Z 300.168,A -85,B 0,C 180,E1 23903.814,E2 23903.814} C_VEL
LIN {X 0,Y 543.412,Z 309.078,A -85,B 0,C 180,E1 23902.546,E2 23902.546} C_VEL
LIN {X 0,Y 554.642,Z 324.652,A -85,B 0,C 180,E1 23900.628,E2 23900.628} C_VEL
LIN {X 0,Y 566.114,Z 341.495,A -85,B 0,C 180,E1 23898.808,E2 23898.808} C_VEL
LIN {X 0,Y 577.776,Z 359.574,A -85,B 0,C 180,E1 23897.079,E2 23897.079} C_VEL
LIN {X 0,Y 580.775,Z 364.602,A -85,B 0,C 180,E1 23896.648,E2 23896.648} C_VEL
LIN {X 0,Y 573.679,Z 578.05,A -85,B 0,C 180,E1 23893.581,E2 23893.581} C_VEL
LIN {X 0,Y 569.257,Z 712.188,A -85,B 0,C 180,E1 23891.658,E2 23891.658} C_VEL
LIN {X 0,Y 567.432,Z 739.319,A -85,B 0,C 180,E1 23891.125,E2 23891.125} C_VEL
LIN {X 0,Y 566.607,Z 749.206,A -85,B 0,C 180,E1 23890.875,E2 23890.875} C_VEL
LIN {X 0,Y 565.201,Z 756.77,A -85,B 0,C 180,E1 23890.741,E2 23890.741} C_VEL
LIN {X 0,Y 559.041,Z 774.798,A -85,B 0,C 180,E1 23890.578,E2 23890.578} C_VEL
LIN {X 0,Y 557.244,Z 782.008,A -85,B 0,C 180,E1 23890.408,E2 23890.408} C_VEL
LIN {X 0,Y 557.101,Z 783.032,A -85,B 0,C 180,E1 23890.373,E2 23890.373} C_VEL
LIN {X 0,Y 553.922,Z 807.357,A -85,B 0,C 180,E1 23889.389,E2 23889.389} C_VEL
LIN {X 0,Y 550.448,Z 829.961,A -85,B 0,C 180,E1 23888.274,E2 23888.274} C_VEL
LIN {X 0,Y 547.197,Z 849.539,A -85,B 0,C 180,E1 23887.151,E2 23887.151} C_VEL
LIN {X 0,Y 543.25,Z 871.606,A -85,B 0,C 180,E1 23885.694,E2 23885.694} C_VEL
LIN {X 0,Y 539.155,Z 892.629,A -85,B 0,C 180,E1 23884.061,E2 23884.061} C_VEL
LIN {X 0,Y 535.662,Z 910.102,A -85,B 0,C 180,E1 23882.52,E2 23882.52} C_VEL
LIN {X 0,Y 531.509,Z 930.528,A -85,B 0,C 180,E1 23880.463,E2 23880.463} C_VEL
LIN {X 0,Y 527.973,Z 947.397,A -85,B 0,C 180,E1 23878.505,E2 23878.505} C_VEL
LIN {X 0,Y 524.801,Z 962.903,A -85,B 0,C 180,E1 23876.476,E2 23876.476} C_VEL
LIN {X 0,Y 521.377,Z 980.217,A -85,B 0,C 180,E1 23873.869,E2 23873.869} C_VEL
LIN {X 0,Y 519.01,Z 992.722,A -85,B 0,C 180,E1 23871.709,E2 23871.709} C_VEL
LIN {X 0,Y 516.935,Z 1004.972,A -85,B 0,C 180,E1 23869.315,E2 23869.315} C_VEL
LIN {X 0,Y 515.015,Z 1017.435,A -85,B 0,C 180,E1 23866.466,E2 23866.466} C_VEL
LIN {X 0,Y 513.897,Z 1025.976,A -85,B 0,C 180,E1 23864.191,E2 23864.191} C_VEL
LIN {X 0,Y 513.035,Z 1034.042,A -85,B 0,C 180,E1 23861.694,E2 23861.694} C_VEL
LIN {X 0,Y 512.407,Z 1041.794,A -85,B 0,C 180,E1 23858.755,E2 23858.755} C_VEL
LIN {X 0,Y 512.108,Z 1046.92,A -85,B 0,C 180,E1 23856.277,E2 23856.277} C_VEL
LIN {X 0,Y 511.977,Z 1050.53,A -85,B 0,C 180,E1 23854.032,E2 23854.032} C_VEL
LIN {X 0,Y 511.905,Z 1053.373,A -85,B 0,C 180,E1 23851.567,E2 23851.567} C_VEL
LIN {X 0,Y 511.9,Z 1055.163,A -85,B 0,C 180,E1 23848.769,E2 23848.769} C_VEL
LIN {X 0,Y 511.898,Z 1055.374,A -85,B 0,C 180,E1 23846.192,E2 23846.192} C_VEL
LIN {X 0,Y 511.916,Z 1054.468,A -85,B 0,C 180,E1 23843.826,E2 23843.826} C_VEL
LIN {X 0,Y 511.923,Z 1052.491,A -85,B 0,C 180,E1 23841.463,E2 23841.463} C_VEL
LIN {X 0,Y 512.038,Z 1048.688,A -85,B 0,C 180,E1 23838.606,E2 23838.606} C_VEL
LIN {X 0,Y 512.292,Z 1043.404,A -85,B 0,C 180,E1 23835.879,E2 23835.879} C_VEL
LIN {X 0,Y 512.693,Z 1037.823,A -85,B 0,C 180,E1 23833.573,E2 23833.573} C_VEL
LIN {X 0,Y 513.367,Z 1030.746,A -85,B 0,C 180,E1 23831.136,E2 23831.136} C_VEL
LIN {X 0,Y 514.598,Z 1020.49,A -85,B 0,C 180,E1 23828.215,E2 23828.215} C_VEL
LIN {X 0,Y 515.997,Z 1010.762,A -85,B 0,C 180,E1 23825.866,E2 23825.866} C_VEL
LIN {X 0,Y 517.814,Z 999.632,A -85,B 0,C 180,E1 23823.509,E2 23823.509} C_VEL
LIN {X 0,Y 520.489,Z 984.785,A -85,B 0,C 180,E1 23820.794,E2 23820.794} C_VEL
LIN {X 0,Y 523.095,Z 971.47,A -85,B 0,C 180,E1 23818.673,E2 23818.673} C_VEL
LIN {X 0,Y 526.192,Z 956.399,A -85,B 0,C 180,E1 23816.534,E2 23816.534} C_VEL
LIN {X 0,Y 530.124,Z 937.516,A -85,B 0,C 180,E1 23814.198,E2 23814.198} C_VEL
LIN {X 0,Y 533.559,Z 921.306,A -85,B 0,C 180,E1 23812.439,E2 23812.439} C_VEL
LIN {X 0,Y 537.679,Z 901.913,A -85,B 0,C 180,E1 23810.575,E2 23810.575} C_VEL
LIN {X 0,Y 541.978,Z 880.479,A -85,B 0,C 180,E1 23808.805,E2 23808.805} C_VEL
LIN {X 0,Y 545.466,Z 862.434,A -85,B 0,C 180,E1 23807.501,E2 23807.501} C_VEL
LIN {X 0,Y 549.156,Z 842.265,A -85,B 0,C 180,E1 23806.22,E2 23806.22} C_VEL
LIN {X 0,Y 553.236,Z 817.476,A -85,B 0,C 180,E1 23804.889,E2 23804.889} C_VEL
LIN {X 0,Y 556.211,Z 797.415,A -85,B 0,C 180,E1 23803.982,E2 23803.982} C_VEL
LIN {X 0,Y 558.813,Z 777.695,A -85,B 0,C 180,E1 23803.223,E2 23803.223} C_VEL
LIN {X 0,Y 561.663,Z 752.403,A -85,B 0,C 180,E1 23802.428,E2 23802.428} C_VEL
LIN {X 0,Y 563.689,Z 728.962,A -85,B 0,C 180,E1 23801.869,E2 23801.869} C_VEL
LIN {X 0,Y 565.036,Z 707.512,A -85,B 0,C 180,E1 23801.479,E2 23801.479} C_VEL
LIN {X 0,Y 573.678,Z 472.321,A -85,B 0,C 180,E1 23798.056,E2 23798.056} C_VEL
LIN {X 0,Y 577.51,Z 368.343,A -85,B 0,C 180,E1 23796.509,E2 23796.509} C_VEL
LIN {X 0,Y 567.329,Z 352.399,A -85,B 0,C 180,E1 23794.853,E2 23794.853} C_VEL
LIN {X 0,Y 556.061,Z 335.876,A -85,B 0,C 180,E1 23792.892,E2 23792.892} C_VEL
LIN {X 0,Y 544.702,Z 320.261,A -85,B 0,C 180,E1 23790.746,E2 23790.746} C_VEL
LIN {X 0,Y 537.393,Z 311.092,A -85,B 0,C 180,E1 23789.267,E2 23789.267} C_VEL
LIN {X 0,Y 533.7,Z 306.432,A -85,B 0,C 180,E1 23788.477,E2 23788.477} C_VEL
LIN {X 0,Y 530.172,Z 302.384,A -85,B 0,C 180,E1 23787.703,E2 23787.703} C_VEL
LIN {X 0,Y 528.904,Z 300.599,A -85,B 0,C 180,E1 23787.409,E2 23787.409} C_VEL
LIN {X 0,Y 525.565,Z 297.143,A -85,B 0,C 180,E1 23786.649,E2 23786.649} C_VEL
LIN {X 0,Y 523.852,Z 294.543,A -85,B 0,C 180,E1 23786.223,E2 23786.223} C_VEL
LIN {X 0,Y 520.61,Z 291.537,A -85,B 0,C 180,E1 23785.451,E2 23785.451} C_VEL
LIN {X 0,Y 518.807,Z 288.46,A -85,B 0,C 180,E1 23784.966,E2 23784.966} C_VEL
LIN {X 0,Y 515.645,Z 286.138,A -85,B 0,C 180,E1 23784.182,E2 23784.182} C_VEL
LIN {X 0,Y 513.899,Z 282.736,A -85,B 0,C 180,E1 23783.592,E2 23783.592} C_VEL
LIN {X 0,Y 513.746,Z 282.011,A -85,B 0,C 180,E1 23783.151,E2 23783.151} C_VEL
LIN {X 0,Y 513.792,Z 281.902,A -85,B 0,C 180,E1 23779.912,E2 23779.912} C_VEL
LIN {X 0,Y 513.755,Z 281.98,A -85,B 0,C 180,E1 23776.508,E2 23776.508} C_VEL
LIN {X 0,Y 513.733,Z 281.908,A -85,B 0,C 180,E1 23773.048,E2 23773.048} C_VEL
LIN {X 0,Y 513.798,Z 281.966,A -85,B 0,C 180,E1 23769.748,E2 23769.748} C_VEL
LIN {X 0,Y 513.737,Z 281.9,A -85,B 0,C 180,E1 23766.482,E2 23766.482} C_VEL
LIN {X 0,Y 513.747,Z 281.979,A -85,B 0,C 180,E1 23763.012,E2 23763.012} C_VEL
LIN {X 0,Y 513.803,Z 281.892,A -85,B 0,C 180,E1 23759.666,E2 23759.666} C_VEL
LIN {X 0,Y 513.753,Z 281.985,A -85,B 0,C 180,E1 23756.206,E2 23756.206} C_VEL
LIN {X 0,Y 513.733,Z 281.898,A -85,B 0,C 180,E1 23752.732,E2 23752.732} C_VEL
LIN {X 0,Y 513.801,Z 281.976,A -85,B 0,C 180,E1 23749.459,E2 23749.459} C_VEL
LIN {X 0,Y 513.742,Z 281.897,A -85,B 0,C 180,E1 23746.034,E2 23746.034} C_VEL
LIN {X 0,Y 513.745,Z 281.979,A -85,B 0,C 180,E1 23742.559,E2 23742.559} C_VEL
LIN {X 0,Y 513.787,Z 281.902,A -85,B 0,C 180,E1 23739.137,E2 23739.137} C_VEL
LIN {X 0,Y 513.753,Z 281.971,A -85,B 0,C 180,E1 23735.876,E2 23735.876} C_VEL
LIN {X 0,Y 513.788,Z 282.243,A -85,B 0,C 180,E1 23733.907,E2 23733.907} C_VEL
LIN {X 0,Y 515.027,Z 285.341,A -85,B 0,C 180,E1 23733.105,E2 23733.105} C_VEL
LIN {X 0,Y 518.286,Z 289.116,A -85,B 0,C 180,E1 23732.231,E2 23732.231} C_VEL
LIN {X 0,Y 522.726,Z 294.338,A -85,B 0,C 180,E1 23731.119,E2 23731.119} C_VEL
LIN {X 0,Y 526.263,Z 298.62,A -85,B 0,C 180,E1 23730.271,E2 23730.271} C_VEL
LIN {X 0,Y 533.148,Z 307.432,A -85,B 0,C 180,E1 23728.701,E2 23728.701} C_VEL
LIN {X 0,Y 540.827,Z 317.412,A -85,B 0,C 180,E1 23727.074,E2 23727.074} C_VEL
LIN {X 0,Y 551.388,Z 331.73,A -85,B 0,C 180,E1 23725.006,E2 23725.006} C_VEL
LIN {X 0,Y 560.818,Z 345.439,A -85,B 0,C 180,E1 23723.293,E2 23723.293} C_VEL
LIN {X 0,Y 571.313,Z 361.325,A -85,B 0,C 180,E1 23721.524,E2 23721.524} C_VEL
LIN {X 0,Y 577.689,Z 371.888,A -85,B 0,C 180,E1 23720.496,E2 23720.496} C_VEL
LIN {X 0,Y 568.967,Z 603.265,A -85,B 0,C 180,E1 23717.119,E2 23717.119} C_VEL
LIN {X 0,Y 564.654,Z 720.187,A -85,B 0,C 180,E1 23715.409,E2 23715.409} C_VEL
LIN {X 0,Y 562.63,Z 747.617,A -85,B 0,C 180,E1 23714.864,E2 23714.864} C_VEL
LIN {X 0,Y 560.336,Z 770.472,A -85,B 0,C 180,E1 23714.244,E2 23714.244} C_VEL
LIN {X 0,Y 557.911,Z 790.92,A -85,B 0,C 180,E1 23713.559,E2 23713.559} C_VEL
LIN {X 0,Y 554.688,Z 814.641,A -85,B 0,C 180,E1 23712.6,E2 23712.6} C_VEL
LIN {X 0,Y 550.954,Z 837.926,A -85,B 0,C 180,E1 23711.45,E2 23711.45} C_VEL
LIN {X 0,Y 547.775,Z 856.402,A -85,B 0,C 180,E1 23710.391,E2 23710.391} C_VEL
LIN {X 0,Y 544.088,Z 876.502,A -85,B 0,C 180,E1 23709.075,E2 23709.075} C_VEL
LIN {X 0,Y 539.618,Z 899.106,A -85,B 0,C 180,E1 23707.352,E2 23707.352} C_VEL
LIN {X 0,Y 535.981,Z 916.908,A -85,B 0,C 180,E1 23705.792,E2 23705.792} C_VEL
LIN {X 0,Y 532.098,Z 935.767,A -85,B 0,C 180,E1 23703.925,E2 23703.925} C_VEL
LIN {X 0,Y 528.129,Z 954.732,A -85,B 0,C 180,E1 23701.758,E2 23701.758} C_VEL
LIN {X 0,Y 525.028,Z 969.827,A -85,B 0,C 180,E1 23699.806,E2 23699.806} C_VEL
LIN {X 0,Y 521.781,Z 986.467,A -85,B 0,C 180,E1 23697.381,E2 23697.381} C_VEL
LIN {X 0,Y 519.087,Z 1000.831,A -85,B 0,C 180,E1 23694.951,E2 23694.951} C_VEL
LIN {X 0,Y 517.113,Z 1012.445,A -85,B 0,C 180,E1 23692.731,E2 23692.731} C_VEL
LIN {X 0,Y 515.286,Z 1024.593,A -85,B 0,C 180,E1 23690.085,E2 23690.085} C_VEL
LIN {X 0,Y 513.937,Z 1034.829,A -85,B 0,C 180,E1 23687.434,E2 23687.434} C_VEL
LIN {X 0,Y 513.128,Z 1042.469,A -85,B 0,C 180,E1 23685.136,E2 23685.136} C_VEL
LIN {X 0,Y 512.506,Z 1049.863,A -85,B 0,C 180,E1 23682.507,E2 23682.507} C_VEL
LIN {X 0,Y 512.125,Z 1056.235,A -85,B 0,C 180,E1 23679.604,E2 23679.604} C_VEL
LIN {X 0,Y 511.987,Z 1060.236,A -85,B 0,C 180,E1 23677.203,E2 23677.203} C_VEL
LIN {X 0,Y 511.917,Z 1062.977,A -85,B 0,C 180,E1 23674.93,E2 23674.93} C_VEL
LIN {X 0,Y 511.906,Z 1064.888,A -85,B 0,C 180,E1 23672.351,E2 23672.351} C_VEL
LIN {X 0,Y 511.896,Z 1065.374,A -85,B 0,C 180,E1 23669.44,E2 23669.44} C_VEL
LIN {X 0,Y 511.914,Z 1064.545,A -85,B 0,C 180,E1 23667.089,E2 23667.089} C_VEL
LIN {X 0,Y 511.922,Z 1062.747,A -85,B 0,C 180,E1 23664.845,E2 23664.845} C_VEL
LIN {X 0,Y 512,Z 1059.785,A -85,B 0,C 180,E1 23662.482,E2 23662.482} C_VEL
LIN {X 0,Y 512.192,Z 1054.831,A -85,B 0,C 180,E1 23659.654,E2 23659.654} C_VEL
LIN {X 0,Y 512.612,Z 1048.339,A -85,B 0,C 180,E1 23656.923,E2 23656.923} C_VEL
LIN {X 0,Y 513.235,Z 1041.405,A -85,B 0,C 180,E1 23654.52,E2 23654.52} C_VEL
LIN {X 0,Y 514.311,Z 1031.973,A -85,B 0,C 180,E1 23651.76,E2 23651.76} C_VEL
LIN {X 0,Y 515.798,Z 1021.007,A -85,B 0,C 180,E1 23649.103,E2 23649.103} C_VEL
LIN {X 0,Y 517.406,Z 1010.639,A -85,B 0,C 180,E1 23646.903,E2 23646.903} C_VEL
LIN {X 0,Y 519.821,Z 997.021,A -85,B 0,C 180,E1 23644.355,E2 23644.355} C_VEL
LIN {X 0,Y 522.717,Z 981.47,A -85,B 0,C 180,E1 23641.865,E2 23641.865} C_VEL
LIN {X 0,Y 525.367,Z 968.089,A -85,B 0,C 180,E1 23639.964,E2 23639.964} C_VEL
LIN {X 0,Y 528.999,Z 950.373,A -85,B 0,C 180,E1 23637.726,E2 23637.726} C_VEL
LIN {X 0,Y 532.689,Z 932.031,A -85,B 0,C 180,E1 23635.729,E2 23635.729} C_VEL
LIN {X 0,Y 536.13,Z 915.038,A -85,B 0,C 180,E1 23634.088,E2 23634.088} C_VEL
LIN {X 0,Y 540.337,Z 893.965,A -85,B 0,C 180,E1 23632.296,E2 23632.296} C_VEL
LIN {X 0,Y 544.16,Z 873.374,A -85,B 0,C 180,E1 23630.795,E2 23630.795} C_VEL
LIN {X 0,Y 547.428,Z 854.881,A -85,B 0,C 180,E1 23629.611,E2 23629.611} C_VEL
LIN {X 0,Y 550.897,Z 833.94,A -85,B 0,C 180,E1 23628.441,E2 23628.441} C_VEL
